LIN {X 0,Y 566.188,Z 287.454,A -85,B 0,C 180,E1 -2641.075,E2 -2641.075} C_VEL
LIN {X 0,Y 566.21,Z 287.455,A -85,B 0,C 180,E1 -2643.733,E2 -2643.733} C_VEL
LIN {X 0,Y 566.179,Z 287.455,A -85,B 0,C 180,E1 -2646.57,E2 -2646.57} C_VEL
LIN {X 0,Y 566.211,Z 287.456,A -85,B 0,C 180,E1 -2649.685,E2 -2649.685} C_VEL
LIN {X 0,Y 566.196,Z 287.452,A -85,B 0,C 180,E1 -2652.916,E2 -2652.916} C_VEL
LIN {X 0,Y 566.193,Z 287.458,A -85,B 0,C 180,E1 -2656.048,E2 -2656.048} C_VEL
LIN {X 0,Y 566.204,Z 287.45,A -85,B 0,C 180,E1 -2658.863,E2 -2658.863} C_VEL
LIN {X 0,Y 566.181,Z 287.46,A -85,B 0,C 180,E1 -2661.636,E2 -2661.636} C_VEL
LIN {X 0,Y 566.158,Z 287.457,A -85,B 0,C 180,E1 -2664.307,E2 -2664.307} C_VEL
LIN {X 0,Y 566.198,Z 287.45,A -85,B 0,C 180,E1 -2666.896,E2 -2666.896} C_VEL
LIN {X 0,Y 566.174,Z 287.46,A -85,B 0,C 180,E1 -2669.406,E2 -2669.406} C_VEL
LIN {X 0,Y 566.221,Z 287.451,A -85,B 0,C 180,E1 -2671.858,E2 -2671.858} C_VEL
LIN {X 0,Y 566.204,Z 287.45,A -85,B 0,C 180,E1 -2674.25,E2 -2674.25} C_VEL
LIN {X 0,Y 566.164,Z 287.456,A -85,B 0,C 180,E1 -2676.717,E2 -2676.717} C_VEL
LIN {X 0,Y 566.211,Z 287.454,A -85,B 0,C 180,E1 -2679.662,E2 -2679.662} C_VEL
LIN {X 0,Y 566.191,Z 287.449,A -85,B 0,C 180,E1 -2682.668,E2 -2682.668} C_VEL
LIN {X 0,Y 566.224,Z 287.454,A -85,B 0,C 180,E1 -2685.626,E2 -2685.626} C_VEL
LIN {X 0,Y 566.266,Z 287.442,A -85,B 0,C 180,E1 -2688.654,E2 -2688.654} C_VEL
LIN {X 0,Y 566.238,Z 287.452,A -85,B 0,C 180,E1 -2691.434,E2 -2691.434} C_VEL
LIN {X 0,Y 566.25,Z 287.444,A -85,B 0,C 180,E1 -2694.301,E2 -2694.301} C_VEL
LIN {X 0,Y 566.265,Z 287.443,A -85,B 0,C 180,E1 -2697.866,E2 -2697.866} C_VEL
LIN {X 0,Y 566.299,Z 287.436,A -85,B 0,C 180,E1 -2700.711,E2 -2700.711} C_VEL
LIN {X 0,Y 566.27,Z 287.445,A -85,B 0,C 180,E1 -2702.845,E2 -2702.845} C_VEL
LIN {X 0,Y 566.249,Z 287.447,A -85,B 0,C 180,E1 -2705.698,E2 -2705.698} C_VEL
LIN {X 0,Y 566.224,Z 287.448,A -85,B 0,C 180,E1 -2708.565,E2 -2708.565} C_VEL
LIN {X 0,Y 566.24,Z 287.448,A -85,B 0,C 180,E1 -2711.454,E2 -2711.454} C_VEL
LIN {X 0,Y 566.223,Z 287.451,A -85,B 0,C 180,E1 -2714.507,E2 -2714.507} C_VEL
LIN {X 0,Y 566.189,Z 287.454,A -85,B 0,C 180,E1 -2717.331,E2 -2717.331} C_VEL
LIN {X 0,Y 566.209,Z 287.448,A -85,B 0,C 180,E1 -2720.337,E2 -2720.337} C_VEL
LIN {X 0,Y 566.179,Z 287.456,A -85,B 0,C 180,E1 -2723.404,E2 -2723.404} C_VEL
LIN {X 0,Y 566.204,Z 287.449,A -85,B 0,C 180,E1 -2725.749,E2 -2725.749} C_VEL
LIN {X 0,Y 566.201,Z 287.449,A -85,B 0,C 180,E1 -2727.497,E2 -2727.497} C_VEL
LIN {X 0,Y 565.527,Z 287.533,A -85,B 0,C 180,E1 -2728.091,E2 -2728.091} C_VEL
LIN {X 0,Y 562.664,Z 287.897,A -85,B 0,C 180,E1 -2729.054,E2 -2729.054} C_VEL
LIN {X 0,Y 560.253,Z 288.195,A -85,B 0,C 180,E1 -2729.83,E2 -2729.83} C_VEL
LIN {X 0,Y 559.224,Z 288.324,A -85,B 0,C 180,E1 -2730.429,E2 -2730.429} C_VEL
LIN {X 0,Y 559.143,Z 288.332,A -85,B 0,C 180,E1 -2730.631,E2 -2730.631} C_VEL
LIN {X 0,Y 559.168,Z 288.325,A -85,B 0,C 180,E1 -2733.574,E2 -2733.574} C_VEL
LIN {X 0,Y 559.16,Z 288.332,A -85,B 0,C 180,E1 -2736.449,E2 -2736.449} C_VEL
LIN {X 0,Y 559.169,Z 288.332,A -85,B 0,C 180,E1 -2738.934,E2 -2738.934} C_VEL
LIN {X 0,Y 559.183,Z 288.324,A -85,B 0,C 180,E1 -2741.768,E2 -2741.768} C_VEL
LIN {X 0,Y 559.131,Z 288.338,A -85,B 0,C 180,E1 -2744.739,E2 -2744.739} C_VEL
LIN {X 0,Y 559.156,Z 288.322,A -85,B 0,C 180,E1 -2747.257,E2 -2747.257} C_VEL
LIN {X 0,Y 559.178,Z 288.326,A -85,B 0,C 180,E1 -2750.135,E2 -2750.135} C_VEL
LIN {X 0,Y 559.139,Z 288.334,A -85,B 0,C 180,E1 -2752.893,E2 -2752.893} C_VEL
LIN {X 0,Y 559.153,Z 288.324,A -85,B 0,C 180,E1 -2755.557,E2 -2755.557} C_VEL
LIN {X 0,Y 559.166,Z 288.333,A -85,B 0,C 180,E1 -2758.138,E2 -2758.138} C_VEL
LIN {X 0,Y 559.138,Z 288.335,A -85,B 0,C 180,E1 -2760.647,E2 -2760.647} C_VEL
LIN {X 0,Y 559.177,Z 288.327,A -85,B 0,C 180,E1 -2763.17,E2 -2763.17} C_VEL
LIN {X 0,Y 559.152,Z 288.33,A -85,B 0,C 180,E1 -2765.495,E2 -2765.495} C_VEL
LIN {X 0,Y 559.167,Z 288.333,A -85,B 0,C 180,E1 -2768.624,E2 -2768.624} C_VEL
LIN {X 0,Y 559.167,Z 288.329,A -85,B 0,C 180,E1 -2770.927,E2 -2770.927} C_VEL
LIN {X 0,Y 559.164,Z 288.334,A -85,B 0,C 180,E1 -2773.948,E2 -2773.948} C_VEL
LIN {X 0,Y 559.169,Z 288.337,A -85,B 0,C 180,E1 -2776.184,E2 -2776.184} C_VEL
LIN {X 0,Y 559.193,Z 288.325,A -85,B 0,C 180,E1 -2779.134,E2 -2779.134} C_VEL
LIN {X 0,Y 559.201,Z 288.333,A -85,B 0,C 180,E1 -2782.054,E2 -2782.054} C_VEL
LIN {X 0,Y 559.251,Z 288.318,A -85,B 0,C 180,E1 -2784.953,E2 -2784.953} C_VEL
LIN {X 0,Y 559.254,Z 288.325,A -85,B 0,C 180,E1 -2787.839,E2 -2787.839} C_VEL
LIN {X 0,Y 559.27,Z 288.317,A -85,B 0,C 180,E1 -2790.72,E2 -2790.72} C_VEL
LIN {X 0,Y 559.235,Z 288.32,A -85,B 0,C 180,E1 -2792.881,E2 -2792.881} C_VEL
LIN {X 0,Y 559.229,Z 288.328,A -85,B 0,C 180,E1 -2795.77,E2 -2795.77} C_VEL
LIN {X 0,Y 559.184,Z 288.327,A -85,B 0,C 180,E1 -2798.674,E2 -2798.674} C_VEL
LIN {X 0,Y 559.202,Z 288.33,A -85,B 0,C 180,E1 -2801.6,E2 -2801.6} C_VEL
LIN {X 0,Y 559.196,Z 288.325,A -85,B 0,C 180,E1 -2804.595,E2 -2804.595} C_VEL
LIN {X 0,Y 559.159,Z 288.336,A -85,B 0,C 180,E1 -2807.556,E2 -2807.556} C_VEL
LIN {X 0,Y 559.168,Z 288.336,A -85,B 0,C 180,E1 -2809.837,E2 -2809.837} C_VEL
LIN {X 0,Y 559.137,Z 288.335,A -85,B 0,C 180,E1 -2812.152,E2 -2812.152} C_VEL
LIN {X 0,Y 559.175,Z 288.33,A -85,B 0,C 180,E1 -2815.187,E2 -2815.187} C_VEL
LIN {X 0,Y 559.189,Z 288.332,A -85,B 0,C 180,E1 -2817.711,E2 -2817.711} C_VEL
LIN {X 0,Y 559.157,Z 288.33,A -85,B 0,C 180,E1 -2821.018,E2 -2821.018} C_VEL
LIN {X 0,Y 559.171,Z 288.325,A -85,B 0,C 180,E1 -2823.951,E2 -2823.951} C_VEL
LIN {X 0,Y 559.162,Z 288.327,A -85,B 0,C 180,E1 -2826.448,E2 -2826.448} C_VEL
LIN {X 0,Y 559.17,Z 288.329,A -85,B 0,C 180,E1 -2828.933,E2 -2828.933} C_VEL
LIN {X 0,Y 559.184,Z 288.322,A -85,B 0,C 180,E1 -2831.767,E2 -2831.767} C_VEL
LIN {X 0,Y 559.131,Z 288.331,A -85,B 0,C 180,E1 -2834.739,E2 -2834.739} C_VEL
LIN {X 0,Y 559.168,Z 288.328,A -85,B 0,C 180,E1 -2837.862,E2 -2837.862} C_VEL
LIN {X 0,Y 559.177,Z 288.325,A -85,B 0,C 180,E1 -2840.135,E2 -2840.135} C_VEL
LIN {X 0,Y 559.138,Z 288.335,A -85,B 0,C 180,E1 -2842.892,E2 -2842.892} C_VEL
LIN {X 0,Y 559.153,Z 288.332,A -85,B 0,C 180,E1 -2845.556,E2 -2845.556} C_VEL
LIN {X 0,Y 559.161,Z 288.328,A -85,B 0,C 180,E1 -2848.138,E2 -2848.138} C_VEL
LIN {X 0,Y 559.148,Z 288.331,A -85,B 0,C 180,E1 -2850.647,E2 -2850.647} C_VEL
LIN {X 0,Y 559.161,Z 288.334,A -85,B 0,C 180,E1 -2853.172,E2 -2853.172} C_VEL
LIN {X 0,Y 559.147,Z 288.334,A -85,B 0,C 180,E1 -2855.495,E2 -2855.495} C_VEL
LIN {X 0,Y 559.166,Z 288.33,A -85,B 0,C 180,E1 -2858.624,E2 -2858.624} C_VEL
LIN {X 0,Y 559.161,Z 288.332,A -85,B 0,C 180,E1 -2860.926,E2 -2860.926} C_VEL
LIN {X 0,Y 559.161,Z 288.328,A -85,B 0,C 180,E1 -2863.948,E2 -2863.948} C_VEL
LIN {X 0,Y 559.164,Z 288.328,A -85,B 0,C 180,E1 -2866.184,E2 -2866.184} C_VEL
LIN {X 0,Y 559.2,Z 288.323,A -85,B 0,C 180,E1 -2869.134,E2 -2869.134} C_VEL
LIN {X 0,Y 559.196,Z 288.321,A -85,B 0,C 180,E1 -2872.054,E2 -2872.054} C_VEL
LIN {X 0,Y 559.249,Z 288.325,A -85,B 0,C 180,E1 -2874.954,E2 -2874.954} C_VEL
LIN {X 0,Y 559.238,Z 288.316,A -85,B 0,C 180,E1 -2877.84,E2 -2877.84} C_VEL
LIN {X 0,Y 559.269,Z 288.317,A -85,B 0,C 180,E1 -2880.72,E2 -2880.72} C_VEL
LIN {X 0,Y 559.234,Z 288.326,A -85,B 0,C 180,E1 -2882.882,E2 -2882.882} C_VEL
LIN {X 0,Y 559.219,Z 288.32,A -85,B 0,C 180,E1 -2885.771,E2 -2885.771} C_VEL
LIN {X 0,Y 559.193,Z 288.327,A -85,B 0,C 180,E1 -2888.675,E2 -2888.675} C_VEL
LIN {X 0,Y 559.2,Z 288.321,A -85,B 0,C 180,E1 -2891.601,E2 -2891.601} C_VEL
LIN {X 0,Y 559.19,Z 288.333,A -85,B 0,C 180,E1 -2894.596,E2 -2894.596} C_VEL
LIN {X 0,Y 559.151,Z 288.325,A -85,B 0,C 180,E1 -2897.558,E2 -2897.558} C_VEL
LIN {X 0,Y 559.166,Z 288.324,A -85,B 0,C 180,E1 -2899.838,E2 -2899.838} C_VEL
LIN {X 0,Y 559.133,Z 288.335,A -85,B 0,C 180,E1 -2902.154,E2 -2902.154} C_VEL
LIN {X 0,Y 559.167,Z 288.325,A -85,B 0,C 180,E1 -2905.299,E2 -2905.299} C_VEL
LIN {X 0,Y 559.185,Z 288.322,A -85,B 0,C 180,E1 -2907.712,E2 -2907.712} C_VEL
LIN {X 0,Y 559.146,Z 288.336,A -85,B 0,C 180,E1 -2910.184,E2 -2910.184} C_VEL
LIN {X 0,Y 559.146,Z 288.331,A -85,B 0,C 180,E1 -2912.716,E2 -2912.716} C_VEL
LIN {X 0,Y 559.123,Z 288.331,A -85,B 0,C 180,E1 -2915.325,E2 -2915.325} C_VEL
LIN {X 0,Y 559.127,Z 288.338,A -85,B 0,C 180,E1 -2918.018,E2 -2918.018} C_VEL
LIN {X 0,Y 559.152,Z 288.33,A -85,B 0,C 180,E1 -2920.813,E2 -2920.813} C_VEL
LIN {X 0,Y 559.142,Z 288.33,A -85,B 0,C 180,E1 -2923.197,E2 -2923.197} C_VEL
LIN {X 0,Y 559.136,Z 288.339,A -85,B 0,C 180,E1 -2926.267,E2 -2926.267} C_VEL
LIN {X 0,Y 559.152,Z 288.325,A -85,B 0,C 180,E1 -2929.188,E2 -2929.188} C_VEL
LIN {X 0,Y 559.127,Z 288.341,A -85,B 0,C 180,E1 -2931.983,E2 -2931.983} C_VEL
LIN {X 0,Y 559.127,Z 288.333,A -85,B 0,C 180,E1 -2934.788,E2 -2934.788} C_VEL
LIN {X 0,Y 559.154,Z 288.33,A -85,B 0,C 180,E1 -2937.365,E2 -2937.365} C_VEL
LIN {X 0,Y 559.146,Z 288.338,A -85,B 0,C 180,E1 -2940.144,E2 -2940.144} C_VEL
LIN {X 0,Y 559.163,Z 288.332,A -85,B 0,C 180,E1 -2943.175,E2 -2943.175} C_VEL
LIN {X 0,Y 559.212,Z 288.44,A -85,B 0,C 180,E1 -2944.807,E2 -2944.807} C_VEL
LIN {X 0,Y 559.948,Z 294.047,A -85,B 0,C 180,E1 -2945.927,E2 -2945.927} C_VEL
LIN {X 0,Y 559.68,Z 309.675,A -85,B 0,C 180,E1 -2948.838,E2 -2948.838} C_VEL
LIN {X 0,Y 559.517,Z 326.41,A -85,B 0,C 180,E1 -2951.888,E2 -2951.888} C_VEL
LIN {X 0,Y 559.299,Z 343.133,A -85,B 0,C 180,E1 -2954.905,E2 -2954.905} C_VEL
LIN {X 0,Y 559.262,Z 348.266,A -85,B 0,C 180,E1 -2955.792,E2 -2955.792} C_VEL
LIN {X 0,Y 559.602,Z 350.542,A -85,B 0,C 180,E1 -2955.868,E2 -2955.868} C_VEL
LIN {X 0,Y 560.311,Z 356.112,A -85,B 0,C 180,E1 -2955.959,E2 -2955.959} C_VEL
LIN {X 0,Y 560.037,Z 454.578,A -85,B 0,C 180,E1 -2957.245,E2 -2957.245} C_VEL
LIN {X 0,Y 559.976,Z 465.719,A -85,B 0,C 180,E1 -2957.497,E2 -2957.497} C_VEL
LIN {X 0,Y 559.814,Z 478.172,A -85,B 0,C 180,E1 -2957.908,E2 -2957.908} C_VEL
LIN {X 0,Y 559.678,Z 490.904,A -85,B 0,C 180,E1 -2958.503,E2 -2958.503} C_VEL
LIN {X 0,Y 559.509,Z 501.475,A -85,B 0,C 180,E1 -2959.14,E2 -2959.14} C_VEL
LIN {X 0,Y 559.379,Z 510.174,A -85,B 0,C 180,E1 -2959.778,E2 -2959.778} C_VEL
LIN {X 0,Y 559.274,Z 517.542,A -85,B 0,C 180,E1 -2960.416,E2 -2960.416} C_VEL
LIN {X 0,Y 559.137,Z 524.73,A -85,B 0,C 180,E1 -2961.143,E2 -2961.143} C_VEL
LIN {X 0,Y 559.052,Z 532.276,A -85,B 0,C 180,E1 -2962.052,E2 -2962.052} C_VEL
LIN {X 0,Y 558.934,Z 538.681,A -85,B 0,C 180,E1 -2962.976,E2 -2962.976} C_VEL
LIN {X 0,Y 558.909,Z 543.8,A -85,B 0,C 180,E1 -2963.864,E2 -2963.864} C_VEL
LIN {X 0,Y 558.798,Z 548.897,A -85,B 0,C 180,E1 -2964.949,E2 -2964.949} C_VEL
LIN {X 0,Y 558.843,Z 552.853,A -85,B 0,C 180,E1 -2966.034,E2 -2966.034} C_VEL
LIN {X 0,Y 558.799,Z 555.774,A -85,B 0,C 180,E1 -2967.116,E2 -2967.116} C_VEL
LIN {X 0,Y 558.746,Z 558.196,A -85,B 0,C 180,E1 -2968.559,E2 -2968.559} C_VEL
LIN {X 0,Y 558.741,Z 558.78,A -85,B 0,C 180,E1 -2969.279,E2 -2969.279} C_VEL
LIN {X 0,Y 558.741,Z 558.78,A -85,B 0,C 180,E1 -2970.721,E2 -2970.721} C_VEL
LIN {X 0,Y 558.746,Z 558.196,A -85,B 0,C 180,E1 -2971.441,E2 -2971.441} C_VEL
LIN {X 0,Y 558.799,Z 555.774,A -85,B 0,C 180,E1 -2972.884,E2 -2972.884} C_VEL
LIN {X 0,Y 558.843,Z 552.853,A -85,B 0,C 180,E1 -2973.966,E2 -2973.966} C_VEL
LIN {X 0,Y 558.798,Z 548.897,A -85,B 0,C 180,E1 -2975.051,E2 -2975.051} C_VEL
LIN {X 0,Y 558.91,Z 543.8,A -85,B 0,C 180,E1 -2976.136,E2 -2976.136} C_VEL
LIN {X 0,Y 558.974,Z 537.416,A -85,B 0,C 180,E1 -2977.223,E2 -2977.223} C_VEL
LIN {X 0,Y 559.093,Z 529.505,A -85,B 0,C 180,E1 -2978.312,E2 -2978.312} C_VEL
LIN {X 0,Y 559.209,Z 521.359,A -85,B 0,C 180,E1 -2979.221,E2 -2979.221} C_VEL
LIN {X 0,Y 559.33,Z 511.306,A -85,B 0,C 180,E1 -2980.131,E2 -2980.131} C_VEL
LIN {X 0,Y 559.499,Z 502.823,A -85,B 0,C 180,E1 -2980.769,E2 -2980.769} C_VEL
LIN {X 0,Y 559.631,Z 493.792,A -85,B 0,C 180,E1 -2981.335,E2 -2981.335} C_VEL
LIN {X 0,Y 559.768,Z 483.593,A -85,B 0,C 180,E1 -2981.854,E2 -2981.854} C_VEL
LIN {X 0,Y 559.863,Z 474.329,A -85,B 0,C 180,E1 -2982.229,E2 -2982.229} C_VEL
LIN {X 0,Y 559.966,Z 463.971,A -85,B 0,C 180,E1 -2982.549,E2 -2982.549} C_VEL
LIN {X 0,Y 560.068,Z 453.247,A -85,B 0,C 180,E1 -2982.777,E2 -2982.777} C_VEL
LIN {X 0,Y 560.236,Z 354.323,A -85,B 0,C 180,E1 -2984.066,E2 -2984.066} C_VEL
LIN {X 0,Y 559.275,Z 348.595,A -85,B 0,C 180,E1 -2984.184,E2 -2984.184} C_VEL
LIN {X 0,Y 559.225,Z 347.169,A -85,B 0,C 180,E1 -2984.371,E2 -2984.371} C_VEL
LIN {X 0,Y 559.444,Z 330.904,A -85,B 0,C 180,E1 -2987.302,E2 -2987.302} C_VEL
LIN {X 0,Y 559.662,Z 313.862,A -85,B 0,C 180,E1 -2990.393,E2 -2990.393} C_VEL
LIN {X 0,Y 559.864,Z 298.427,A -85,B 0,C 180,E1 -2993.255,E2 -2993.255} C_VEL
LIN {X 0,Y 559.822,Z 291.989,A -85,B 0,C 180,E1 -2994.473,E2 -2994.473} C_VEL
LIN {X 0,Y 559.189,Z 288.353,A -85,B 0,C 180,E1 -2995.251,E2 -2995.251} C_VEL
LIN {X 0,Y 559.138,Z 288.339,A -85,B 0,C 180,E1 -2997.714,E2 -2997.714} C_VEL
LIN {X 0,Y 559.151,Z 288.338,A -85,B 0,C 180,E1 -3000.182,E2 -3000.182} C_VEL
LIN {X 0,Y 559.155,Z 288.329,A -85,B 0,C 180,E1 -3002.714,E2 -3002.714} C_VEL
LIN {X 0,Y 559.121,Z 288.334,A -85,B 0,C 180,E1 -3005.324,E2 -3005.324} C_VEL
LIN {X 0,Y 559.127,Z 288.341,A -85,B 0,C 180,E1 -3008.017,E2 -3008.017} C_VEL
LIN {X 0,Y 559.152,Z 288.325,A -85,B 0,C 180,E1 -3010.812,E2 -3010.812} C_VEL
LIN {X 0,Y 559.136,Z 288.339,A -85,B 0,C 180,E1 -3013.733,E2 -3013.733} C_VEL
LIN {X 0,Y 559.142,Z 288.33,A -85,B 0,C 180,E1 -3016.803,E2 -3016.803} C_VEL
LIN {X 0,Y 559.171,Z 288.328,A -85,B 0,C 180,E1 -3019.188,E2 -3019.188} C_VEL
LIN {X 0,Y 559.127,Z 288.338,A -85,B 0,C 180,E1 -3021.982,E2 -3021.982} C_VEL
LIN {X 0,Y 559.127,Z 288.331,A -85,B 0,C 180,E1 -3024.786,E2 -3024.786} C_VEL
LIN {X 0,Y 559.148,Z 288.332,A -85,B 0,C 180,E1 -3027.364,E2 -3027.364} C_VEL
LIN {X 0,Y 559.141,Z 288.333,A -85,B 0,C 180,E1 -3030.142,E2 -3030.142} C_VEL
LIN {X 0,Y 559.163,Z 288.327,A -85,B 0,C 180,E1 -3033.097,E2 -3033.097} C_VEL
LIN {X 0,Y 559.148,Z 288.336,A -85,B 0,C 180,E1 -3035.494,E2 -3035.494} C_VEL
LIN {X 0,Y 559.169,Z 288.326,A -85,B 0,C 180,E1 -3038.623,E2 -3038.623} C_VEL
LIN {X 0,Y 559.161,Z 288.326,A -85,B 0,C 180,E1 -3040.926,E2 -3040.926} C_VEL
LIN {X 0,Y 559.161,Z 288.33,A -85,B 0,C 180,E1 -3043.947,E2 -3043.947} C_VEL
LIN {X 0,Y 559.165,Z 288.327,A -85,B 0,C 180,E1 -3046.184,E2 -3046.184} C_VEL
LIN {X 0,Y 559.2,Z 288.327,A -85,B 0,C 180,E1 -3049.133,E2 -3049.133} C_VEL
LIN {X 0,Y 559.2,Z 288.321,A -85,B 0,C 180,E1 -3052.053,E2 -3052.053} C_VEL
LIN {X 0,Y 559.249,Z 288.321,A -85,B 0,C 180,E1 -3054.953,E2 -3054.953} C_VEL
LIN {X 0,Y 559.237,Z 288.318,A -85,B 0,C 180,E1 -3057.839,E2 -3057.839} C_VEL
LIN {X 0,Y 559.268,Z 288.311,A -85,B 0,C 180,E1 -3060.72,E2 -3060.72} C_VEL
LIN {X 0,Y 559.236,Z 288.321,A -85,B 0,C 180,E1 -3062.881,E2 -3062.881} C_VEL
LIN {X 0,Y 559.218,Z 288.322,A -85,B 0,C 180,E1 -3065.77,E2 -3065.77} C_VEL
LIN {X 0,Y 559.182,Z 288.326,A -85,B 0,C 180,E1 -3068.674,E2 -3068.674} C_VEL
LIN {X 0,Y 559.198,Z 288.324,A -85,B 0,C 180,E1 -3071.6,E2 -3071.6} C_VEL
LIN {X 0,Y 559.188,Z 288.328,A -85,B 0,C 180,E1 -3074.595,E2 -3074.595} C_VEL
LIN {X 0,Y 559.149,Z 288.328,A -85,B 0,C 180,E1 -3077.557,E2 -3077.557} C_VEL
LIN {X 0,Y 559.164,Z 288.324,A -85,B 0,C 180,E1 -3079.837,E2 -3079.837} C_VEL
LIN {X 0,Y 559.132,Z 288.331,A -85,B 0,C 180,E1 -3082.153,E2 -3082.153} C_VEL
LIN {X 0,Y 559.168,Z 288.33,A -85,B 0,C 180,E1 -3085.187,E2 -3085.187} C_VEL
LIN {X 0,Y 559.181,Z 288.322,A -85,B 0,C 180,E1 -3087.712,E2 -3087.712} C_VEL
LIN {X 0,Y 559.143,Z 288.332,A -85,B 0,C 180,E1 -3090.631,E2 -3090.631} C_VEL
LIN {X 0,Y 558.481,Z 288.418,A -85,B 0,C 180,E1 -3091.233,E2 -3091.233} C_VEL
LIN {X 0,Y 555.617,Z 288.773,A -85,B 0,C 180,E1 -3092.209,E2 -3092.209} C_VEL
LIN {X 0,Y 553.206,Z 289.074,A -85,B 0,C 180,E1 -3092.995,E2 -3092.995} C_VEL
LIN {X 0,Y 552.187,Z 289.195,A -85,B 0,C 180,E1 -3093.601,E2 -3093.601} C_VEL
LIN {X 0,Y 552.114,Z 289.203,A -85,B 0,C 180,E1 -3093.807,E2 -3093.807} C_VEL
LIN {X 0,Y 552.102,Z 289.217,A -85,B 0,C 180,E1 -3096.747,E2 -3096.747} C_VEL
LIN {X 0,Y 552.126,Z 289.203,A -85,B 0,C 180,E1 -3099.527,E2 -3099.527} C_VEL
LIN {X 0,Y 552.122,Z 289.21,A -85,B 0,C 180,E1 -3102.426,E2 -3102.426} C_VEL
LIN {X 0,Y 552.091,Z 289.207,A -85,B 0,C 180,E1 -3105.563,E2 -3105.563} C_VEL
LIN {X 0,Y 552.132,Z 289.205,A -85,B 0,C 180,E1 -3108.676,E2 -3108.676} C_VEL
LIN {X 0,Y 552.112,Z 289.207,A -85,B 0,C 180,E1 -3111.412,E2 -3111.412} C_VEL
LIN {X 0,Y 552.106,Z 289.211,A -85,B 0,C 180,E1 -3114.159,E2 -3114.159} C_VEL
LIN {X 0,Y 552.123,Z 289.209,A -85,B 0,C 180,E1 -3116.816,E2 -3116.816} C_VEL
LIN {X 0,Y 552.102,Z 289.207,A -85,B 0,C 180,E1 -3119.391,E2 -3119.391} C_VEL
LIN {X 0,Y 552.121,Z 289.206,A -85,B 0,C 180,E1 -3121.903,E2 -3121.903} C_VEL
LIN {X 0,Y 552.152,Z 289.207,A -85,B 0,C 180,E1 -3124.649,E2 -3124.649} C_VEL
LIN {X 0,Y 552.091,Z 289.21,A -85,B 0,C 180,E1 -3127.55,E2 -3127.55} C_VEL
LIN {X 0,Y 552.153,Z 289.206,A -85,B 0,C 180,E1 -3130.675,E2 -3130.675} C_VEL
LIN {X 0,Y 552.114,Z 289.21,A -85,B 0,C 180,E1 -3133.738,E2 -3133.738} C_VEL
LIN {X 0,Y 552.132,Z 289.212,A -85,B 0,C 180,E1 -3136.005,E2 -3136.005} C_VEL
LIN {X 0,Y 552.16,Z 289.202,A -85,B 0,C 180,E1 -3138.994,E2 -3138.994} C_VEL
LIN {X 0,Y 552.155,Z 289.21,A -85,B 0,C 180,E1 -3141.952,E2 -3141.952} C_VEL
LIN {X 0,Y 552.226,Z 289.194,A -85,B 0,C 180,E1 -3144.889,E2 -3144.889} C_VEL
LIN {X 0,Y 552.224,Z 289.2,A -85,B 0,C 180,E1 -3147.812,E2 -3147.812} C_VEL
LIN {X 0,Y 552.24,Z 289.193,A -85,B 0,C 180,E1 -3150.729,E2 -3150.729} C_VEL
LIN {X 0,Y 552.202,Z 289.197,A -85,B 0,C 180,E1 -3152.918,E2 -3152.918} C_VEL
LIN {X 0,Y 552.199,Z 289.205,A -85,B 0,C 180,E1 -3155.844,E2 -3155.844} C_VEL
LIN {X 0,Y 552.156,Z 289.202,A -85,B 0,C 180,E1 -3158.786,E2 -3158.786} C_VEL
LIN {X 0,Y 552.159,Z 289.209,A -85,B 0,C 180,E1 -3161.75,E2 -3161.75} C_VEL
LIN {X 0,Y 552.133,Z 289.205,A -85,B 0,C 180,E1 -3164.748,E2 -3164.748} C_VEL
LIN {X 0,Y 552.111,Z 289.216,A -85,B 0,C 180,E1 -3167.788,E2 -3167.788} C_VEL
LIN {X 0,Y 552.127,Z 289.209,A -85,B 0,C 180,E1 -3170.101,E2 -3170.101} C_VEL
LIN {X 0,Y 552.091,Z 289.21,A -85,B 0,C 180,E1 -3172.45,E2 -3172.45} C_VEL
LIN {X 0,Y 552.152,Z 289.207,A -85,B 0,C 180,E1 -3175.351,E2 -3175.351} C_VEL
LIN {X 0,Y 552.121,Z 289.206,A -85,B 0,C 180,E1 -3178.097,E2 -3178.097} C_VEL
LIN {X 0,Y 552.102,Z 289.207,A -85,B 0,C 180,E1 -3180.609,E2 -3180.609} C_VEL
LIN {X 0,Y 552.123,Z 289.209,A -85,B 0,C 180,E1 -3183.184,E2 -3183.184} C_VEL
LIN {X 0,Y 552.106,Z 289.211,A -85,B 0,C 180,E1 -3185.841,E2 -3185.841} C_VEL
LIN {X 0,Y 552.118,Z 289.209,A -85,B 0,C 180,E1 -3189.062,E2 -3189.062} C_VEL
LIN {X 0,Y 552.132,Z 289.203,A -85,B 0,C 180,E1 -3191.444,E2 -3191.444} C_VEL
LIN {X 0,Y 552.088,Z 289.207,A -85,B 0,C 180,E1 -3194.532,E2 -3194.532} C_VEL
LIN {X 0,Y 552.122,Z 289.21,A -85,B 0,C 180,E1 -3197.584,E2 -3197.584} C_VEL
LIN {X 0,Y 552.126,Z 289.203,A -85,B 0,C 180,E1 -3200.473,E2 -3200.473} C_VEL
LIN {X 0,Y 552.105,Z 289.215,A -85,B 0,C 180,E1 -3203.315,E2 -3203.315} C_VEL
LIN {X 0,Y 552.131,Z 289.202,A -85,B 0,C 180,E1 -3205.94,E2 -3205.94} C_VEL
LIN {X 0,Y 552.108,Z 289.208,A -85,B 0,C 180,E1 -3208.54,E2 -3208.54} C_VEL
LIN {X 0,Y 552.117,Z 289.207,A -85,B 0,C 180,E1 -3211.437,E2 -3211.437} C_VEL
LIN {X 0,Y 552.119,Z 289.204,A -85,B 0,C 180,E1 -3214.356,E2 -3214.356} C_VEL
LIN {X 0,Y 552.1,Z 289.212,A -85,B 0,C 180,E1 -3216.758,E2 -3216.758} C_VEL
LIN {X 0,Y 552.117,Z 289.21,A -85,B 0,C 180,E1 -3219.12,E2 -3219.12} C_VEL
LIN {X 0,Y 552.121,Z 289.205,A -85,B 0,C 180,E1 -3221.445,E2 -3221.445} C_VEL
LIN {X 0,Y 552.111,Z 289.206,A -85,B 0,C 180,E1 -3223.738,E2 -3223.738} C_VEL
LIN {X 0,Y 552.126,Z 289.204,A -85,B 0,C 180,E1 -3226.005,E2 -3226.005} C_VEL
LIN {X 0,Y 552.168,Z 289.201,A -85,B 0,C 180,E1 -3228.994,E2 -3228.994} C_VEL
LIN {X 0,Y 552.15,Z 289.199,A -85,B 0,C 180,E1 -3231.952,E2 -3231.952} C_VEL
LIN {X 0,Y 552.223,Z 289.201,A -85,B 0,C 180,E1 -3234.889,E2 -3234.889} C_VEL
LIN {X 0,Y 552.211,Z 289.191,A -85,B 0,C 180,E1 -3237.812,E2 -3237.812} C_VEL
LIN {X 0,Y 552.239,Z 289.192,A -85,B 0,C 180,E1 -3240.73,E2 -3240.73} C_VEL
LIN {X 0,Y 552.2,Z 289.202,A -85,B 0,C 180,E1 -3242.919,E2 -3242.919} C_VEL
LIN {X 0,Y 552.189,Z 289.196,A -85,B 0,C 180,E1 -3245.844,E2 -3245.844} C_VEL
LIN {X 0,Y 552.161,Z 289.2,A -85,B 0,C 180,E1 -3248.786,E2 -3248.786} C_VEL
LIN {X 0,Y 552.155,Z 289.198,A -85,B 0,C 180,E1 -3251.751,E2 -3251.751} C_VEL
LIN {X 0,Y 552.127,Z 289.21,A -85,B 0,C 180,E1 -3254.749,E2 -3254.749} C_VEL
LIN {X 0,Y 552.102,Z 289.204,A -85,B 0,C 180,E1 -3257.789,E2 -3257.789} C_VEL
LIN {X 0,Y 552.126,Z 289.204,A -85,B 0,C 180,E1 -3260.102,E2 -3260.102} C_VEL
LIN {X 0,Y 552.084,Z 289.218,A -85,B 0,C 180,E1 -3262.452,E2 -3262.452} C_VEL
LIN {X 0,Y 552.147,Z 289.199,A -85,B 0,C 180,E1 -3265.351,E2 -3265.351} C_VEL
LIN {X 0,Y 552.119,Z 289.206,A -85,B 0,C 180,E1 -3268.098,E2 -3268.098} C_VEL
LIN {X 0,Y 552.095,Z 289.214,A -85,B 0,C 180,E1 -3270.61,E2 -3270.61} C_VEL
LIN {X 0,Y 552.1,Z 289.205,A -85,B 0,C 180,E1 -3273.187,E2 -3273.187} C_VEL
LIN {X 0,Y 552.08,Z 289.212,A -85,B 0,C 180,E1 -3275.844,E2 -3275.844} C_VEL
LIN {X 0,Y 552.112,Z 289.209,A -85,B 0,C 180,E1 -3278.59,E2 -3278.59} C_VEL
LIN {X 0,Y 552.125,Z 289.205,A -85,B 0,C 180,E1 -3281.446,E2 -3281.446} C_VEL
LIN {X 0,Y 552.089,Z 289.213,A -85,B 0,C 180,E1 -3284.532,E2 -3284.532} C_VEL
LIN {X 0,Y 552.126,Z 289.207,A -85,B 0,C 180,E1 -3287.586,E2 -3287.586} C_VEL
LIN {X 0,Y 552.126,Z 289.208,A -85,B 0,C 180,E1 -3290.474,E2 -3290.474} C_VEL
LIN {X 0,Y 552.096,Z 289.209,A -85,B 0,C 180,E1 -3293.319,E2 -3293.319} C_VEL
LIN {X 0,Y 552.124,Z 289.213,A -85,B 0,C 180,E1 -3295.94,E2 -3295.94} C_VEL
LIN {X 0,Y 552.119,Z 289.209,A -85,B 0,C 180,E1 -3298.541,E2 -3298.541} C_VEL
LIN {X 0,Y 552.104,Z 289.212,A -85,B 0,C 180,E1 -3301.443,E2 -3301.443} C_VEL
LIN {X 0,Y 552.126,Z 289.212,A -85,B 0,C 180,E1 -3304.356,E2 -3304.356} C_VEL
LIN {X 0,Y 552.163,Z 289.447,A -85,B 0,C 180,E1 -3304.686,E2 -3304.686} C_VEL
LIN {X 0,Y 553.01,Z 294.996,A -85,B 0,C 180,E1 -3305.805,E2 -3305.805} C_VEL
LIN {X 0,Y 552.706,Z 310.587,A -85,B 0,C 180,E1 -3308.753,E2 -3308.753} C_VEL
LIN {X 0,Y 552.501,Z 327.322,A -85,B 0,C 180,E1 -3311.842,E2 -3311.842} C_VEL
LIN {X 0,Y 552.283,Z 344.026,A -85,B 0,C 180,E1 -3314.879,E2 -3314.879} C_VEL
LIN {X 0,Y 552.236,Z 348.45,A -85,B 0,C 180,E1 -3315.622,E2 -3315.622} C_VEL
LIN {X 0,Y 553.424,Z 355.602,A -85,B 0,C 180,E1 -3315.773,E2 -3315.773} C_VEL
LIN {X 0,Y 553.139,Z 453.191,A -85,B 0,C 180,E1 -3317.06,E2 -3317.06} C_VEL
LIN {X 0,Y 553.051,Z 463.937,A -85,B 0,C 180,E1 -3317.291,E2 -3317.291} C_VEL
LIN {X 0,Y 552.925,Z 474.306,A -85,B 0,C 180,E1 -3317.615,E2 -3317.615} C_VEL
LIN {X 0,Y 552.767,Z 484.372,A -85,B 0,C 180,E1 -3318.03,E2 -3318.03} C_VEL
LIN {X 0,Y 552.636,Z 494.743,A -85,B 0,C 180,E1 -3318.575,E2 -3318.575} C_VEL
LIN {X 0,Y 552.469,Z 505.496,A -85,B 0,C 180,E1 -3319.278,E2 -3319.278} C_VEL
LIN {X 0,Y 552.272,Z 515.616,A -85,B 0,C 180,E1 -3320.108,E2 -3320.108} C_VEL
LIN {X 0,Y 552.122,Z 524.721,A -85,B 0,C 180,E1 -3321.029,E2 -3321.029} C_VEL
LIN {X 0,Y 551.984,Z 532.268,A -85,B 0,C 180,E1 -3321.949,E2 -3321.949} C_VEL
LIN {X 0,Y 551.886,Z 538.557,A -85,B 0,C 180,E1 -3322.868,E2 -3322.868} C_VEL
LIN {X 0,Y 551.836,Z 544.396,A -85,B 0,C 180,E1 -3323.902,E2 -3323.902} C_VEL
LIN {X 0,Y 551.739,Z 550.388,A -85,B 0,C 180,E1 -3325.251,E2 -3325.251} C_VEL
LIN {X 0,Y 551.75,Z 553.976,A -85,B 0,C 180,E1 -3326.349,E2 -3326.349} C_VEL
LIN {X 0,Y 551.723,Z 555.768,A -85,B 0,C 180,E1 -3327.079,E2 -3327.079} C_VEL
LIN {X 0,Y 551.645,Z 558.195,A -85,B 0,C 180,E1 -3328.54,E2 -3328.54} C_VEL
LIN {X 0,Y 551.641,Z 558.779,A -85,B 0,C 180,E1 -3329.27,E2 -3329.27} C_VEL
LIN {X 0,Y 551.641,Z 558.779,A -85,B 0,C 180,E1 -3330.73,E2 -3330.73} C_VEL
LIN {X 0,Y 551.645,Z 558.195,A -85,B 0,C 180,E1 -3331.46,E2 -3331.46} C_VEL
LIN {X 0,Y 551.723,Z 555.768,A -85,B 0,C 180,E1 -3332.921,E2 -3332.921} C_VEL
LIN {X 0,Y 551.764,Z 552.845,A -85,B 0,C 180,E1 -3334.017,E2 -3334.017} C_VEL
LIN {X 0,Y 551.723,Z 548.888,A -85,B 0,C 180,E1 -3335.116,E2 -3335.116} C_VEL
LIN {X 0,Y 551.836,Z 544.395,A -85,B 0,C 180,E1 -3336.098,E2 -3336.098} C_VEL
LIN {X 0,Y 551.886,Z 538.557,A -85,B 0,C 180,E1 -3337.132,E2 -3337.132} C_VEL
LIN {X 0,Y 551.984,Z 532.268,A -85,B 0,C 180,E1 -3338.051,E2 -3338.051} C_VEL
LIN {X 0,Y 552.122,Z 524.721,A -85,B 0,C 180,E1 -3338.971,E2 -3338.971} C_VEL
LIN {X 0,Y 552.272,Z 515.616,A -85,B 0,C 180,E1 -3339.892,E2 -3339.892} C_VEL
LIN {X 0,Y 552.489,Z 504.156,A -85,B 0,C 180,E1 -3340.814,E2 -3340.814} C_VEL
LIN {X 0,Y 552.632,Z 494.762,A -85,B 0,C 180,E1 -3341.424,E2 -3341.424} C_VEL
LIN {X 0,Y 552.794,Z 484.679,A -85,B 0,C 180,E1 -3341.955,E2 -3341.955} C_VEL
LIN {X 0,Y 552.881,Z 475.596,A -85,B 0,C 180,E1 -3342.34,E2 -3342.34} C_VEL
LIN {X 0,Y 553.054,Z 464.811,A -85,B 0,C 180,E1 -3342.685,E2 -3342.685} C_VEL
LIN {X 0,Y 553.131,Z 454.522,A -85,B 0,C 180,E1 -3342.917,E2 -3342.917} C_VEL
LIN {X 0,Y 553.343,Z 369.327,A -85,B 0,C 180,E1 -3344.049,E2 -3344.049} C_VEL
LIN {X 0,Y 553.316,Z 354.796,A -85,B 0,C 180,E1 -3344.24,E2 -3344.24} C_VEL
LIN {X 0,Y 552.236,Z 348.447,A -85,B 0,C 180,E1 -3344.378,E2 -3344.378} C_VEL
LIN {X 0,Y 552.283,Z 344.026,A -85,B 0,C 180,E1 -3345.121,E2 -3345.121} C_VEL
LIN {X 0,Y 552.501,Z 327.322,A -85,B 0,C 180,E1 -3348.158,E2 -3348.158} C_VEL
LIN {X 0,Y 552.706,Z 310.619,A -85,B 0,C 180,E1 -3351.247,E2 -3351.247} C_VEL
LIN {X 0,Y 552.99,Z 295.021,A -85,B 0,C 180,E1 -3354.196,E2 -3354.196} C_VEL
LIN {X 0,Y 552.151,Z 289.247,A -85,B 0,C 180,E1 -3355.385,E2 -3355.385} C_VEL
LIN {X 0,Y 552.088,Z 289.217,A -85,B 0,C 180,E1 -3358.099,E2 -3358.099} C_VEL
LIN {X 0,Y 552.1,Z 289.211,A -85,B 0,C 180,E1 -3360.609,E2 -3360.609} C_VEL
LIN {X 0,Y 552.114,Z 289.206,A -85,B 0,C 180,E1 -3363.185,E2 -3363.185} C_VEL
LIN {X 0,Y 552.072,Z 289.217,A -85,B 0,C 180,E1 -3365.844,E2 -3365.844} C_VEL
LIN {X 0,Y 552.113,Z 289.207,A -85,B 0,C 180,E1 -3368.588,E2 -3368.588} C_VEL
LIN {X 0,Y 552.116,Z 289.204,A -85,B 0,C 180,E1 -3371.445,E2 -3371.445} C_VEL
LIN {X 0,Y 552.088,Z 289.21,A -85,B 0,C 180,E1 -3374.531,E2 -3374.531} C_VEL
LIN {X 0,Y 552.127,Z 289.21,A -85,B 0,C 180,E1 -3377.584,E2 -3377.584} C_VEL
LIN {X 0,Y 552.125,Z 289.204,A -85,B 0,C 180,E1 -3380.472,E2 -3380.472} C_VEL
LIN {X 0,Y 552.1,Z 289.211,A -85,B 0,C 180,E1 -3383.316,E2 -3383.316} C_VEL
LIN {X 0,Y 552.098,Z 289.211,A -85,B 0,C 180,E1 -3385.937,E2 -3385.937} C_VEL
LIN {X 0,Y 552.112,Z 289.206,A -85,B 0,C 180,E1 -3388.54,E2 -3388.54} C_VEL
LIN {X 0,Y 552.119,Z 289.212,A -85,B 0,C 180,E1 -3391.437,E2 -3391.437} C_VEL
LIN {X 0,Y 552.122,Z 289.203,A -85,B 0,C 180,E1 -3394.355,E2 -3394.355} C_VEL
LIN {X 0,Y 552.09,Z 289.209,A -85,B 0,C 180,E1 -3396.757,E2 -3396.757} C_VEL
LIN {X 0,Y 552.118,Z 289.208,A -85,B 0,C 180,E1 -3399.119,E2 -3399.119} C_VEL
LIN {X 0,Y 552.119,Z 289.208,A -85,B 0,C 180,E1 -3401.444,E2 -3401.444} C_VEL
LIN {X 0,Y 552.111,Z 289.21,A -85,B 0,C 180,E1 -3403.737,E2 -3403.737} C_VEL
LIN {X 0,Y 552.128,Z 289.205,A -85,B 0,C 180,E1 -3406.004,E2 -3406.004} C_VEL
LIN {X 0,Y 552.168,Z 289.2,A -85,B 0,C 180,E1 -3408.993,E2 -3408.993} C_VEL
LIN {X 0,Y 552.154,Z 289.199,A -85,B 0,C 180,E1 -3411.951,E2 -3411.951} C_VEL
LIN {X 0,Y 552.223,Z 289.196,A -85,B 0,C 180,E1 -3414.889,E2 -3414.889} C_VEL
LIN {X 0,Y 552.21,Z 289.193,A -85,B 0,C 180,E1 -3417.811,E2 -3417.811} C_VEL
LIN {X 0,Y 552.238,Z 289.186,A -85,B 0,C 180,E1 -3420.729,E2 -3420.729} C_VEL
LIN {X 0,Y 552.202,Z 289.197,A -85,B 0,C 180,E1 -3422.918,E2 -3422.918} C_VEL
LIN {X 0,Y 552.188,Z 289.197,A -85,B 0,C 180,E1 -3425.844,E2 -3425.844} C_VEL
LIN {X 0,Y 552.153,Z 289.203,A -85,B 0,C 180,E1 -3428.785,E2 -3428.785} C_VEL
LIN {X 0,Y 552.154,Z 289.2,A -85,B 0,C 180,E1 -3431.75,E2 -3431.75} C_VEL
LIN {X 0,Y 552.126,Z 289.21,A -85,B 0,C 180,E1 -3434.748,E2 -3434.748} C_VEL
LIN {X 0,Y 552.1,Z 289.204,A -85,B 0,C 180,E1 -3437.788,E2 -3437.788} C_VEL
LIN {X 0,Y 552.123,Z 289.201,A -85,B 0,C 180,E1 -3440.101,E2 -3440.101} C_VEL
LIN {X 0,Y 552.086,Z 289.211,A -85,B 0,C 180,E1 -3442.451,E2 -3442.451} C_VEL
LIN {X 0,Y 552.144,Z 289.203,A -85,B 0,C 180,E1 -3445.351,E2 -3445.351} C_VEL
LIN {X 0,Y 552.115,Z 289.202,A -85,B 0,C 180,E1 -3448.097,E2 -3448.097} C_VEL
LIN {X 0,Y 552.103,Z 289.213,A -85,B 0,C 180,E1 -3450.627,E2 -3450.627} C_VEL
LIN {X 0,Y 552.119,Z 289.206,A -85,B 0,C 180,E1 -3453.185,E2 -3453.185} C_VEL
LIN {X 0,Y 552.114,Z 289.203,A -85,B 0,C 180,E1 -3453.807,E2 -3453.807} C_VEL
LIN {X 0,Y 551.48,Z 289.288,A -85,B 0,C 180,E1 -3454.415,E2 -3454.415} C_VEL
LIN {X 0,Y 548.654,Z 289.645,A -85,B 0,C 180,E1 -3455.403,E2 -3455.403} C_VEL
LIN {X 0,Y 546.228,Z 289.951,A -85,B 0,C 180,E1 -3456.199,E2 -3456.199} C_VEL
LIN {X 0,Y 545.157,Z 290.081,A -85,B 0,C 180,E1 -3456.813,E2 -3456.813} C_VEL
LIN {X 0,Y 545.055,Z 290.091,A -85,B 0,C 180,E1 -3457.021,E2 -3457.021} C_VEL
LIN {X 0,Y 545.084,Z 290.082,A -85,B 0,C 180,E1 -3460.14,E2 -3460.14} C_VEL
LIN {X 0,Y 545.069,Z 290.087,A -85,B 0,C 180,E1 -3463.107,E2 -3463.107} C_VEL
LIN {X 0,Y 545.056,Z 290.087,A -85,B 0,C 180,E1 -3466.225,E2 -3466.225} C_VEL
LIN {X 0,Y 545.089,Z 290.082,A -85,B 0,C 180,E1 -3468.887,E2 -3468.887} C_VEL
LIN {X 0,Y 545.046,Z 290.087,A -85,B 0,C 180,E1 -3471.763,E2 -3471.763} C_VEL
LIN {X 0,Y 545.058,Z 290.087,A -85,B 0,C 180,E1 -3474.534,E2 -3474.534} C_VEL
LIN {X 0,Y 545.077,Z 290.083,A -85,B 0,C 180,E1 -3477.213,E2 -3477.213} C_VEL
LIN {X 0,Y 545.06,Z 290.086,A -85,B 0,C 180,E1 -3479.811,E2 -3479.811} C_VEL
LIN {X 0,Y 545.091,Z 290.089,A -85,B 0,C 180,E1 -3482.345,E2 -3482.345} C_VEL
LIN {X 0,Y 545.113,Z 290.082,A -85,B 0,C 180,E1 -3484.821,E2 -3484.821} C_VEL
LIN {X 0,Y 545.039,Z 290.089,A -85,B 0,C 180,E1 -3487.243,E2 -3487.243} C_VEL
LIN {X 0,Y 545.116,Z 290.086,A -85,B 0,C 180,E1 -3490.415,E2 -3490.415} C_VEL
LIN {X 0,Y 545.07,Z 290.086,A -85,B 0,C 180,E1 -3493.521,E2 -3493.521} C_VEL
LIN {X 0,Y 545.091,Z 290.086,A -85,B 0,C 180,E1 -3495.82,E2 -3495.82} C_VEL
LIN {X 0,Y 545.115,Z 290.08,A -85,B 0,C 180,E1 -3498.85,E2 -3498.85} C_VEL
LIN {X 0,Y 545.126,Z 290.084,A -85,B 0,C 180,E1 -3501.847,E2 -3501.847} C_VEL
LIN {X 0,Y 545.202,Z 290.069,A -85,B 0,C 180,E1 -3504.823,E2 -3504.823} C_VEL
LIN {X 0,Y 545.196,Z 290.075,A -85,B 0,C 180,E1 -3507.784,E2 -3507.784} C_VEL
LIN {X 0,Y 545.21,Z 290.068,A -85,B 0,C 180,E1 -3510.739,E2 -3510.739} C_VEL
LIN {X 0,Y 545.169,Z 290.073,A -85,B 0,C 180,E1 -3512.956,E2 -3512.956} C_VEL
LIN {X 0,Y 545.171,Z 290.08,A -85,B 0,C 180,E1 -3515.919,E2 -3515.919} C_VEL
LIN {X 0,Y 545.115,Z 290.08,A -85,B 0,C 180,E1 -3518.9,E2 -3518.9} C_VEL
LIN {X 0,Y 545.131,Z 290.085,A -85,B 0,C 180,E1 -3521.904,E2 -3521.904} C_VEL
LIN {X 0,Y 545.082,Z 290.084,A -85,B 0,C 180,E1 -3524.943,E2 -3524.943} C_VEL
LIN {X 0,Y 545.079,Z 290.089,A -85,B 0,C 180,E1 -3528.025,E2 -3528.025} C_VEL
LIN {X 0,Y 545.091,Z 290.083,A -85,B 0,C 180,E1 -3530.372,E2 -3530.372} C_VEL
LIN {X 0,Y 545.086,Z 290.09,A -85,B 0,C 180,E1 -3533.558,E2 -3533.558} C_VEL
LIN {X 0,Y 545.084,Z 290.087,A -85,B 0,C 180,E1 -3536,E2 -3536} C_VEL
LIN {X 0,Y 545.085,Z 290.08,A -85,B 0,C 180,E1 -3538.748,E2 -3538.748} C_VEL
LIN {X 0,Y 545.072,Z 290.091,A -85,B 0,C 180,E1 -3541.682,E2 -3541.682} C_VEL
LIN {X 0,Y 545.077,Z 290.076,A -85,B 0,C 180,E1 -3544.562,E2 -3544.562} C_VEL
LIN {X 0,Y 545.033,Z 290.094,A -85,B 0,C 180,E1 -3547.303,E2 -3547.303} C_VEL
LIN {X 0,Y 545.067,Z 290.081,A -85,B 0,C 180,E1 -3550.141,E2 -3550.141} C_VEL
LIN {X 0,Y 545.078,Z 290.077,A -85,B 0,C 180,E1 -3553.105,E2 -3553.105} C_VEL
LIN {X 0,Y 545.058,Z 290.085,A -85,B 0,C 180,E1 -3556.224,E2 -3556.224} C_VEL
LIN {X 0,Y 545.092,Z 290.082,A -85,B 0,C 180,E1 -3558.887,E2 -3558.887} C_VEL
LIN {X 0,Y 545.045,Z 290.09,A -85,B 0,C 180,E1 -3561.763,E2 -3561.763} C_VEL
LIN {X 0,Y 545.056,Z 290.084,A -85,B 0,C 180,E1 -3564.534,E2 -3564.534} C_VEL
LIN {X 0,Y 545.073,Z 290.09,A -85,B 0,C 180,E1 -3567.212,E2 -3567.212} C_VEL
LIN {X 0,Y 545.092,Z 290.082,A -85,B 0,C 180,E1 -3569.813,E2 -3569.813} C_VEL
LIN {X 0,Y 545.086,Z 290.082,A -85,B 0,C 180,E1 -3572.826,E2 -3572.826} C_VEL
LIN {X 0,Y 545.042,Z 290.089,A -85,B 0,C 180,E1 -3575.631,E2 -3575.631} C_VEL
LIN {X 0,Y 545.059,Z 290.09,A -85,B 0,C 180,E1 -3578.837,E2 -3578.837} C_VEL
LIN {X 0,Y 545.074,Z 290.086,A -85,B 0,C 180,E1 -3581.196,E2 -3581.196} C_VEL
LIN {X 0,Y 545.067,Z 290.086,A -85,B 0,C 180,E1 -3583.521,E2 -3583.521} C_VEL
LIN {X 0,Y 545.085,Z 290.082,A -85,B 0,C 180,E1 -3585.82,E2 -3585.82} C_VEL
LIN {X 0,Y 545.122,Z 290.081,A -85,B 0,C 180,E1 -3588.85,E2 -3588.85} C_VEL
LIN {X 0,Y 545.12,Z 290.074,A -85,B 0,C 180,E1 -3591.847,E2 -3591.847} C_VEL
LIN {X 0,Y 545.198,Z 290.077,A -85,B 0,C 180,E1 -3594.823,E2 -3594.823} C_VEL
LIN {X 0,Y 545.183,Z 290.066,A -85,B 0,C 180,E1 -3597.784,E2 -3597.784} C_VEL
LIN {X 0,Y 545.208,Z 290.067,A -85,B 0,C 180,E1 -3600.739,E2 -3600.739} C_VEL
LIN {X 0,Y 545.166,Z 290.077,A -85,B 0,C 180,E1 -3602.956,E2 -3602.956} C_VEL
LIN {X 0,Y 545.16,Z 290.072,A -85,B 0,C 180,E1 -3605.92,E2 -3605.92} C_VEL
LIN {X 0,Y 545.118,Z 290.075,A -85,B 0,C 180,E1 -3608.9,E2 -3608.9} C_VEL
LIN {X 0,Y 545.127,Z 290.074,A -85,B 0,C 180,E1 -3611.905,E2 -3611.905} C_VEL
LIN {X 0,Y 545.076,Z 290.085,A -85,B 0,C 180,E1 -3614.944,E2 -3614.944} C_VEL
LIN {X 0,Y 545.071,Z 290.081,A -85,B 0,C 180,E1 -3618.026,E2 -3618.026} C_VEL
LIN {X 0,Y 545.091,Z 290.084,A -85,B 0,C 180,E1 -3620.373,E2 -3620.373} C_VEL
LIN {X 0,Y 545.073,Z 290.083,A -85,B 0,C 180,E1 -3623.56,E2 -3623.56} C_VEL
LIN {X 0,Y 545.072,Z 290.084,A -85,B 0,C 180,E1 -3626.001,E2 -3626.001} C_VEL
LIN {X 0,Y 545.083,Z 290.085,A -85,B 0,C 180,E1 -3628.749,E2 -3628.749} C_VEL
LIN {X 0,Y 545.05,Z 290.087,A -85,B 0,C 180,E1 -3631.68,E2 -3631.68} C_VEL
LIN {X 0,Y 545.054,Z 290.089,A -85,B 0,C 180,E1 -3634.565,E2 -3634.565} C_VEL
LIN {X 0,Y 545.03,Z 290.089,A -85,B 0,C 180,E1 -3637.305,E2 -3637.305} C_VEL
LIN {X 0,Y 545.06,Z 290.09,A -85,B 0,C 180,E1 -3640.144,E2 -3640.144} C_VEL
LIN {X 0,Y 545.074,Z 290.083,A -85,B 0,C 180,E1 -3643.107,E2 -3643.107} C_VEL
LIN {X 0,Y 545.046,Z 290.095,A -85,B 0,C 180,E1 -3646.227,E2 -3646.227} C_VEL
LIN {X 0,Y 545.077,Z 290.078,A -85,B 0,C 180,E1 -3648.886,E2 -3648.886} C_VEL
LIN {X 0,Y 545.076,Z 290.083,A -85,B 0,C 180,E1 -3650.819,E2 -3650.819} C_VEL
LIN {X 0,Y 545.032,Z 290.091,A -85,B 0,C 180,E1 -3653.62,E2 -3653.62} C_VEL
LIN {X 0,Y 545.064,Z 290.089,A -85,B 0,C 180,E1 -3656.329,E2 -3656.329} C_VEL
LIN {X 0,Y 545.065,Z 290.086,A -85,B 0,C 180,E1 -3658.953,E2 -3658.953} C_VEL
LIN {X 0,Y 545.082,Z 290.088,A -85,B 0,C 180,E1 -3661.507,E2 -3661.507} C_VEL
LIN {X 0,Y 545.117,Z 290.204,A -85,B 0,C 180,E1 -3664.487,E2 -3664.487} C_VEL
LIN {X 0,Y 546.05,Z 295.944,A -85,B 0,C 180,E1 -3665.679,E2 -3665.679} C_VEL
LIN {X 0,Y 545.72,Z 311.498,A -85,B 0,C 180,E1 -3668.666,E2 -3668.666} C_VEL
LIN {X 0,Y 545.488,Z 328.233,A -85,B 0,C 180,E1 -3671.794,E2 -3671.794} C_VEL
LIN {X 0,Y 545.239,Z 344.935,A -85,B 0,C 180,E1 -3674.87,E2 -3674.87} C_VEL
LIN {X 0,Y 545.18,Z 348.282,A -85,B 0,C 180,E1 -3675.434,E2 -3675.434} C_VEL
LIN {X 0,Y 546.547,Z 357.582,A -85,B 0,C 180,E1 -3675.619,E2 -3675.619} C_VEL
LIN {X 0,Y 546.242,Z 453.069,A -85,B 0,C 180,E1 -3676.894,E2 -3676.894} C_VEL
LIN {X 0,Y 546.135,Z 462.962,A -85,B 0,C 180,E1 -3677.104,E2 -3677.104} C_VEL
LIN {X 0,Y 546.013,Z 472.938,A -85,B 0,C 180,E1 -3677.408,E2 -3677.408} C_VEL
LIN {X 0,Y 545.853,Z 482.296,A -85,B 0,C 180,E1 -3677.782,E2 -3677.782} C_VEL
LIN {X 0,Y 545.685,Z 492.48,A -85,B 0,C 180,E1 -3678.299,E2 -3678.299} C_VEL
LIN {X 0,Y 545.549,Z 501.441,A -85,B 0,C 180,E1 -3678.859,E2 -3678.859} C_VEL
LIN {X 0,Y 545.392,Z 510.148,A -85,B 0,C 180,E1 -3679.513,E2 -3679.513} C_VEL
LIN {X 0,Y 545.221,Z 517.519,A -85,B 0,C 180,E1 -3680.166,E2 -3680.166} C_VEL
LIN {X 0,Y 545.099,Z 524.713,A -85,B 0,C 180,E1 -3680.913,E2 -3680.913} C_VEL
LIN {X 0,Y 544.973,Z 530.889,A -85,B 0,C 180,E1 -3681.658,E2 -3681.658} C_VEL
LIN {X 0,Y 544.836,Z 537.397,A -85,B 0,C 180,E1 -3682.589,E2 -3682.589} C_VEL
LIN {X 0,Y 544.76,Z 542.262,A -85,B 0,C 180,E1 -3683.408,E2 -3683.408} C_VEL
LIN {X 0,Y 544.738,Z 547.335,A -85,B 0,C 180,E1 -3684.447,E2 -3684.447} C_VEL
LIN {X 0,Y 544.664,Z 551.63,A -85,B 0,C 180,E1 -3685.56,E2 -3685.56} C_VEL
LIN {X 0,Y 544.669,Z 553.974,A -85,B 0,C 180,E1 -3686.301,E2 -3686.301} C_VEL
LIN {X 0,Y 544.65,Z 555.762,A -85,B 0,C 180,E1 -3687.041,E2 -3687.041} C_VEL
LIN {X 0,Y 544.546,Z 558.189,A -85,B 0,C 180,E1 -3688.521,E2 -3688.521} C_VEL
LIN {X 0,Y 544.542,Z 558.772,A -85,B 0,C 180,E1 -3689.261,E2 -3689.261} C_VEL
LIN {X 0,Y 544.542,Z 558.772,A -85,B 0,C 180,E1 -3690.739,E2 -3690.739} C_VEL
LIN {X 0,Y 544.546,Z 558.189,A -85,B 0,C 180,E1 -3691.479,E2 -3691.479} C_VEL
LIN {X 0,Y 544.65,Z 555.762,A -85,B 0,C 180,E1 -3692.959,E2 -3692.959} C_VEL
LIN {X 0,Y 544.684,Z 552.838,A -85,B 0,C 180,E1 -3694.069,E2 -3694.069} C_VEL
LIN {X 0,Y 544.653,Z 548.879,A -85,B 0,C 180,E1 -3695.182,E2 -3695.182} C_VEL
LIN {X 0,Y 544.759,Z 544.638,A -85,B 0,C 180,E1 -3696.128,E2 -3696.128} C_VEL
LIN {X 0,Y 544.79,Z 539.697,A -85,B 0,C 180,E1 -3697.039,E2 -3697.039} C_VEL
LIN {X 0,Y 544.916,Z 533.63,A -85,B 0,C 180,E1 -3697.969,E2 -3697.969} C_VEL
LIN {X 0,Y 545.038,Z 526.333,A -85,B 0,C 180,E1 -3698.901,E2 -3698.901} C_VEL
LIN {X 0,Y 545.198,Z 519.432,A -85,B 0,C 180,E1 -3699.647,E2 -3699.647} C_VEL
LIN {X 0,Y 545.349,Z 511.279,A -85,B 0,C 180,E1 -3700.394,E2 -3700.394} C_VEL
LIN {X 0,Y 545.525,Z 502.791,A -85,B 0,C 180,E1 -3701.048,E2 -3701.048} C_VEL
LIN {X 0,Y 545.699,Z 493.465,A -85,B 0,C 180,E1 -3701.644,E2 -3701.644} C_VEL
LIN {X 0,Y 545.84,Z 483.304,A -85,B 0,C 180,E1 -3702.171,E2 -3702.171} C_VEL
LIN {X 0,Y 545.986,Z 474.226,A -85,B 0,C 180,E1 -3702.545,E2 -3702.545} C_VEL
LIN {X 0,Y 546.128,Z 464.711,A -85,B 0,C 180,E1 -3702.849,E2 -3702.849} C_VEL
LIN {X 0,Y 546.208,Z 454.4,A -85,B 0,C 180,E1 -3703.084,E2 -3703.084} C_VEL
LIN {X 0,Y 546.417,Z 398.906,A -85,B 0,C 180,E1 -3703.836,E2 -3703.836} C_VEL
LIN {X 0,Y 546.401,Z 355.337,A -85,B 0,C 180,E1 -3704.415,E2 -3704.415} C_VEL
LIN {X 0,Y 545.18,Z 348.279,A -85,B 0,C 180,E1 -3704.566,E2 -3704.566} C_VEL
LIN {X 0,Y 545.303,Z 338.676,A -85,B 0,C 180,E1 -3706.279,E2 -3706.279} C_VEL
LIN {X 0,Y 545.489,Z 324.051,A -85,B 0,C 180,E1 -3708.984,E2 -3708.984} C_VEL
LIN {X 0,Y 545.776,Z 309.467,A -85,B 0,C 180,E1 -3711.728,E2 -3711.728} C_VEL
LIN {X 0,Y 546.046,Z 295.97,A -85,B 0,C 180,E1 -3714.321,E2 -3714.321} C_VEL
LIN {X 0,Y 545.092,Z 290.115,A -85,B 0,C 180,E1 -3715.555,E2 -3715.555} C_VEL
LIN {X 0,Y 545.082,Z 290.088,A -85,B 0,C 180,E1 -3718.493,E2 -3718.493} C_VEL
LIN {X 0,Y 545.065,Z 290.086,A -85,B 0,C 180,E1 -3721.047,E2 -3721.047} C_VEL
LIN {X 0,Y 545.064,Z 290.089,A -85,B 0,C 180,E1 -3723.671,E2 -3723.671} C_VEL
LIN {X 0,Y 545.063,Z 290.084,A -85,B 0,C 180,E1 -3726.924,E2 -3726.924} C_VEL
LIN {X 0,Y 545.062,Z 290.085,A -85,B 0,C 180,E1 -3730.142,E2 -3730.142} C_VEL
LIN {X 0,Y 545.075,Z 290.084,A -85,B 0,C 180,E1 -3733.106,E2 -3733.106} C_VEL
LIN {X 0,Y 545.046,Z 290.09,A -85,B 0,C 180,E1 -3736.225,E2 -3736.225} C_VEL
LIN {X 0,Y 545.091,Z 290.08,A -85,B 0,C 180,E1 -3738.886,E2 -3738.886} C_VEL
LIN {X 0,Y 545.047,Z 290.095,A -85,B 0,C 180,E1 -3741.762,E2 -3741.762} C_VEL
LIN {X 0,Y 545.031,Z 290.087,A -85,B 0,C 180,E1 -3744.531,E2 -3744.531} C_VEL
LIN {X 0,Y 545.059,Z 290.085,A -85,B 0,C 180,E1 -3747.21,E2 -3747.21} C_VEL
LIN {X 0,Y 545.056,Z 290.091,A -85,B 0,C 180,E1 -3749.81,E2 -3749.81} C_VEL
LIN {X 0,Y 545.086,Z 290.078,A -85,B 0,C 180,E1 -3752.344,E2 -3752.344} C_VEL
LIN {X 0,Y 545.109,Z 290.076,A -85,B 0,C 180,E1 -3754.82,E2 -3754.82} C_VEL
LIN {X 0,Y 545.03,Z 290.093,A -85,B 0,C 180,E1 -3757.242,E2 -3757.242} C_VEL
LIN {X 0,Y 545.113,Z 290.073,A -85,B 0,C 180,E1 -3760.414,E2 -3760.414} C_VEL
LIN {X 0,Y 545.067,Z 290.09,A -85,B 0,C 180,E1 -3763.521,E2 -3763.521} C_VEL
LIN {X 0,Y 545.087,Z 290.084,A -85,B 0,C 180,E1 -3765.819,E2 -3765.819} C_VEL
LIN {X 0,Y 545.122,Z 290.076,A -85,B 0,C 180,E1 -3768.849,E2 -3768.849} C_VEL
LIN {X 0,Y 545.125,Z 290.076,A -85,B 0,C 180,E1 -3771.847,E2 -3771.847} C_VEL
LIN {X 0,Y 545.198,Z 290.07,A -85,B 0,C 180,E1 -3774.822,E2 -3774.822} C_VEL
LIN {X 0,Y 545.182,Z 290.069,A -85,B 0,C 180,E1 -3777.783,E2 -3777.783} C_VEL
LIN {X 0,Y 545.207,Z 290.061,A -85,B 0,C 180,E1 -3780.738,E2 -3780.738} C_VEL
LIN {X 0,Y 545.168,Z 290.074,A -85,B 0,C 180,E1 -3782.955,E2 -3782.955} C_VEL
LIN {X 0,Y 545.16,Z 290.072,A -85,B 0,C 180,E1 -3785.919,E2 -3785.919} C_VEL
LIN {X 0,Y 545.112,Z 290.081,A -85,B 0,C 180,E1 -3788.9,E2 -3788.9} C_VEL
LIN {X 0,Y 545.125,Z 290.074,A -85,B 0,C 180,E1 -3791.904,E2 -3791.904} C_VEL
LIN {X 0,Y 545.075,Z 290.091,A -85,B 0,C 180,E1 -3794.943,E2 -3794.943} C_VEL
LIN {X 0,Y 545.068,Z 290.08,A -85,B 0,C 180,E1 -3798.026,E2 -3798.026} C_VEL
LIN {X 0,Y 545.088,Z 290.078,A -85,B 0,C 180,E1 -3800.372,E2 -3800.372} C_VEL
LIN {X 0,Y 545.081,Z 290.083,A -85,B 0,C 180,E1 -3803.559,E2 -3803.559} C_VEL
LIN {X 0,Y 545.069,Z 290.081,A -85,B 0,C 180,E1 -3806.001,E2 -3806.001} C_VEL
LIN {X 0,Y 545.083,Z 290.086,A -85,B 0,C 180,E1 -3808.749,E2 -3808.749} C_VEL
LIN {X 0,Y 545.068,Z 290.084,A -85,B 0,C 180,E1 -3811.683,E2 -3811.683} C_VEL
LIN {X 0,Y 545.075,Z 290.087,A -85,B 0,C 180,E1 -3814.563,E2 -3814.563} C_VEL
LIN {X 0,Y 545.055,Z 290.091,A -85,B 0,C 180,E1 -3817.021,E2 -3817.021} C_VEL
LIN {X 0,Y 544.35,Z 290.176,A -85,B 0,C 180,E1 -3817.637,E2 -3817.637} C_VEL
LIN {X 0,Y 541.496,Z 290.538,A -85,B 0,C 180,E1 -3818.638,E2 -3818.638} C_VEL
LIN {X 0,Y 539.119,Z 290.828,A -85,B 0,C 180,E1 -3819.444,E2 -3819.444} C_VEL
LIN {X 0,Y 538.114,Z 290.95,A -85,B 0,C 180,E1 -3820.066,E2 -3820.066} C_VEL
LIN {X 0,Y 538.039,Z 290.959,A -85,B 0,C 180,E1 -3820.277,E2 -3820.277} C_VEL
LIN {X 0,Y 538.017,Z 290.967,A -85,B 0,C 180,E1 -3822.988,E2 -3822.988} C_VEL
LIN {X 0,Y 538.02,Z 290.96,A -85,B 0,C 180,E1 -3825.926,E2 -3825.926} C_VEL
LIN {X 0,Y 538.044,Z 290.956,A -85,B 0,C 180,E1 -3829.225,E2 -3829.225} C_VEL
LIN {X 0,Y 537.987,Z 290.97,A -85,B 0,C 180,E1 -3832.123,E2 -3832.123} C_VEL
LIN {X 0,Y 538.014,Z 290.958,A -85,B 0,C 180,E1 -3834.918,E2 -3834.918} C_VEL
LIN {X 0,Y 538.026,Z 290.961,A -85,B 0,C 180,E1 -3837.619,E2 -3837.619} C_VEL
LIN {X 0,Y 538.013,Z 290.967,A -85,B 0,C 180,E1 -3840.239,E2 -3840.239} C_VEL
LIN {X 0,Y 538.066,Z 290.96,A -85,B 0,C 180,E1 -3842.797,E2 -3842.797} C_VEL
LIN {X 0,Y 538.044,Z 290.96,A -85,B 0,C 180,E1 -3845.293,E2 -3845.293} C_VEL
LIN {X 0,Y 538.01,Z 290.97,A -85,B 0,C 180,E1 -3848.042,E2 -3848.042} C_VEL
LIN {X 0,Y 538.036,Z 290.962,A -85,B 0,C 180,E1 -3850.94,E2 -3850.94} C_VEL
LIN {X 0,Y 538.021,Z 290.963,A -85,B 0,C 180,E1 -3853.299,E2 -3853.299} C_VEL
LIN {X 0,Y 538.06,Z 290.96,A -85,B 0,C 180,E1 -3855.631,E2 -3855.631} C_VEL
LIN {X 0,Y 538.074,Z 290.959,A -85,B 0,C 180,E1 -3858.702,E2 -3858.702} C_VEL
LIN {X 0,Y 538.083,Z 290.96,A -85,B 0,C 180,E1 -3861.74,E2 -3861.74} C_VEL
LIN {X 0,Y 538.16,Z 290.947,A -85,B 0,C 180,E1 -3864.755,E2 -3864.755} C_VEL
LIN {X 0,Y 538.167,Z 290.951,A -85,B 0,C 180,E1 -3867.755,E2 -3867.755} C_VEL
LIN {X 0,Y 538.18,Z 290.944,A -85,B 0,C 180,E1 -3870.748,E2 -3870.748} C_VEL
LIN {X 0,Y 538.136,Z 290.949,A -85,B 0,C 180,E1 -3872.994,E2 -3872.994} C_VEL
LIN {X 0,Y 538.123,Z 290.958,A -85,B 0,C 180,E1 -3875.997,E2 -3875.997} C_VEL
LIN {X 0,Y 538.066,Z 290.958,A -85,B 0,C 180,E1 -3879.017,E2 -3879.017} C_VEL
LIN {X 0,Y 538.08,Z 290.962,A -85,B 0,C 180,E1 -3882.062,E2 -3882.062} C_VEL
LIN {X 0,Y 538.041,Z 290.962,A -85,B 0,C 180,E1 -3885.143,E2 -3885.143} C_VEL
LIN {X 0,Y 538.031,Z 290.964,A -85,B 0,C 180,E1 -3888.27,E2 -3888.27} C_VEL
LIN {X 0,Y 538.035,Z 290.961,A -85,B 0,C 180,E1 -3890.651,E2 -3890.651} C_VEL
LIN {X 0,Y 538.019,Z 290.969,A -85,B 0,C 180,E1 -3893.887,E2 -3893.887} C_VEL
LIN {X 0,Y 538.045,Z 290.96,A -85,B 0,C 180,E1 -3896.366,E2 -3896.366} C_VEL
LIN {X 0,Y 538.026,Z 290.96,A -85,B 0,C 180,E1 -3898.933,E2 -3898.933} C_VEL
LIN {X 0,Y 538.022,Z 290.966,A -85,B 0,C 180,E1 -3901.89,E2 -3901.89} C_VEL
LIN {X 0,Y 538.027,Z 290.954,A -85,B 0,C 180,E1 -3904.621,E2 -3904.621} C_VEL
LIN {X 0,Y 538.001,Z 290.968,A -85,B 0,C 180,E1 -3907.17,E2 -3907.17} C_VEL
LIN {X 0,Y 538.022,Z 290.962,A -85,B 0,C 180,E1 -3909.796,E2 -3909.796} C_VEL
LIN {X 0,Y 538.015,Z 290.953,A -85,B 0,C 180,E1 -3912.785,E2 -3912.785} C_VEL
LIN {X 0,Y 538.021,Z 290.964,A -85,B 0,C 180,E1 -3915.925,E2 -3915.925} C_VEL
LIN {X 0,Y 538.069,Z 290.961,A -85,B 0,C 180,E1 -3919.249,E2 -3919.249} C_VEL
LIN {X 0,Y 537.985,Z 290.967,A -85,B 0,C 180,E1 -3922.122,E2 -3922.122} C_VEL
LIN {X 0,Y 538.012,Z 290.965,A -85,B 0,C 180,E1 -3924.917,E2 -3924.917} C_VEL
LIN {X 0,Y 538.022,Z 290.965,A -85,B 0,C 180,E1 -3927.618,E2 -3927.618} C_VEL
LIN {X 0,Y 538.033,Z 290.96,A -85,B 0,C 180,E1 -3930.24,E2 -3930.24} C_VEL
LIN {X 0,Y 538.056,Z 290.956,A -85,B 0,C 180,E1 -3932.796,E2 -3932.796} C_VEL
LIN {X 0,Y 538.039,Z 290.966,A -85,B 0,C 180,E1 -3935.293,E2 -3935.293} C_VEL
LIN {X 0,Y 538.004,Z 290.963,A -85,B 0,C 180,E1 -3938.042,E2 -3938.042} C_VEL
LIN {X 0,Y 538.03,Z 290.961,A -85,B 0,C 180,E1 -3940.94,E2 -3940.94} C_VEL
LIN {X 0,Y 538.018,Z 290.966,A -85,B 0,C 180,E1 -3943.299,E2 -3943.299} C_VEL
LIN {X 0,Y 538.053,Z 290.959,A -85,B 0,C 180,E1 -3945.631,E2 -3945.631} C_VEL
LIN {X 0,Y 538.079,Z 290.957,A -85,B 0,C 180,E1 -3948.702,E2 -3948.702} C_VEL
LIN {X 0,Y 538.077,Z 290.951,A -85,B 0,C 180,E1 -3951.74,E2 -3951.74} C_VEL
LIN {X 0,Y 538.154,Z 290.953,A -85,B 0,C 180,E1 -3954.755,E2 -3954.755} C_VEL
LIN {X 0,Y 538.155,Z 290.941,A -85,B 0,C 180,E1 -3957.755,E2 -3957.755} C_VEL
LIN {X 0,Y 538.178,Z 290.942,A -85,B 0,C 180,E1 -3960.749,E2 -3960.749} C_VEL
LIN {X 0,Y 538.132,Z 290.953,A -85,B 0,C 180,E1 -3962.995,E2 -3962.995} C_VEL
LIN {X 0,Y 538.113,Z 290.951,A -85,B 0,C 180,E1 -3965.998,E2 -3965.998} C_VEL
LIN {X 0,Y 538.067,Z 290.951,A -85,B 0,C 180,E1 -3969.018,E2 -3969.018} C_VEL
LIN {X 0,Y 538.075,Z 290.954,A -85,B 0,C 180,E1 -3972.063,E2 -3972.063} C_VEL
LIN {X 0,Y 538.036,Z 290.96,A -85,B 0,C 180,E1 -3975.144,E2 -3975.144} C_VEL
LIN {X 0,Y 538.024,Z 290.961,A -85,B 0,C 180,E1 -3978.271,E2 -3978.271} C_VEL
LIN {X 0,Y 538.034,Z 290.966,A -85,B 0,C 180,E1 -3980.652,E2 -3980.652} C_VEL
LIN {X 0,Y 537.996,Z 290.966,A -85,B 0,C 180,E1 -3983.889,E2 -3983.889} C_VEL
LIN {X 0,Y 538.035,Z 290.963,A -85,B 0,C 180,E1 -3986.367,E2 -3986.367} C_VEL
LIN {X 0,Y 538.024,Z 290.963,A -85,B 0,C 180,E1 -3988.934,E2 -3988.934} C_VEL
LIN {X 0,Y 538.003,Z 290.967,A -85,B 0,C 180,E1 -3991.888,E2 -3991.888} C_VEL
LIN {X 0,Y 538.004,Z 290.966,A -85,B 0,C 180,E1 -3994.618,E2 -3994.618} C_VEL
LIN {X 0,Y 537.998,Z 290.965,A -85,B 0,C 180,E1 -3997.171,E2 -3997.171} C_VEL
LIN {X 0,Y 538.017,Z 290.963,A -85,B 0,C 180,E1 -3999.798,E2 -3999.798} C_VEL
LIN {X 0,Y 538.015,Z 290.964,A -85,B 0,C 180,E1 -4002.787,E2 -4002.787} C_VEL
LIN {X 0,Y 538.016,Z 290.968,A -85,B 0,C 180,E1 -4005.927,E2 -4005.927} C_VEL
LIN {X 0,Y 538.045,Z 290.953,A -85,B 0,C 180,E1 -4009.225,E2 -4009.225} C_VEL
LIN {X 0,Y 537.986,Z 290.974,A -85,B 0,C 180,E1 -4012.123,E2 -4012.123} C_VEL
LIN {X 0,Y 537.993,Z 290.965,A -85,B 0,C 180,E1 -4014.916,E2 -4014.916} C_VEL
LIN {X 0,Y 538.017,Z 290.966,A -85,B 0,C 180,E1 -4017.618,E2 -4017.618} C_VEL
LIN {X 0,Y 538.013,Z 290.969,A -85,B 0,C 180,E1 -4020.239,E2 -4020.239} C_VEL
LIN {X 0,Y 538.048,Z 290.963,A -85,B 0,C 180,E1 -4022.796,E2 -4022.796} C_VEL
LIN {X 0,Y 538.084,Z 291.075,A -85,B 0,C 180,E1 -4024.319,E2 -4024.319} C_VEL
LIN {X 0,Y 539.106,Z 297.456,A -85,B 0,C 180,E1 -4025.662,E2 -4025.662} C_VEL
LIN {X 0,Y 538.75,Z 312.423,A -85,B 0,C 180,E1 -4028.577,E2 -4028.577} C_VEL
LIN {X 0,Y 538.466,Z 329.144,A -85,B 0,C 180,E1 -4031.746,E2 -4031.746} C_VEL
LIN {X 0,Y 538.196,Z 345.8,A -85,B 0,C 180,E1 -4034.861,E2 -4034.861} C_VEL
LIN {X 0,Y 538.137,Z 348.086,A -85,B 0,C 180,E1 -4035.24,E2 -4035.24} C_VEL
LIN {X 0,Y 539.677,Z 358.023,A -85,B 0,C 180,E1 -4035.441,E2 -4035.441} C_VEL
LIN {X 0,Y 539.332,Z 452.875,A -85,B 0,C 180,E1 -4036.723,E2 -4036.723} C_VEL
LIN {X 0,Y 539.192,Z 462.767,A -85,B 0,C 180,E1 -4036.935,E2 -4036.935} C_VEL
LIN {X 0,Y 539.093,Z 472.745,A -85,B 0,C 180,E1 -4037.244,E2 -4037.244} C_VEL
LIN {X 0,Y 538.898,Z 482.102,A -85,B 0,C 180,E1 -4037.622,E2 -4037.622} C_VEL
LIN {X 0,Y 538.739,Z 492.047,A -85,B 0,C 180,E1 -4038.132,E2 -4038.132} C_VEL
LIN {X 0,Y 538.549,Z 501.247,A -85,B 0,C 180,E1 -4038.712,E2 -4038.712} C_VEL
LIN {X 0,Y 538.366,Z 509.978,A -85,B 0,C 180,E1 -4039.375,E2 -4039.375} C_VEL
LIN {X 0,Y 538.189,Z 517.375,A -85,B 0,C 180,E1 -4040.036,E2 -4040.036} C_VEL
LIN {X 0,Y 538.055,Z 524.597,A -85,B 0,C 180,E1 -4040.793,E2 -4040.793} C_VEL
LIN {X 0,Y 537.913,Z 530.799,A -85,B 0,C 180,E1 -4041.548,E2 -4041.548} C_VEL
LIN {X 0,Y 537.772,Z 537.335,A -85,B 0,C 180,E1 -4042.491,E2 -4042.491} C_VEL
LIN {X 0,Y 537.673,Z 542.724,A -85,B 0,C 180,E1 -4043.419,E2 -4043.419} C_VEL
LIN {X 0,Y 537.673,Z 547.323,A -85,B 0,C 180,E1 -4044.374,E2 -4044.374} C_VEL
LIN {X 0,Y 537.562,Z 551.622,A -85,B 0,C 180,E1 -4045.501,E2 -4045.501} C_VEL
LIN {X 0,Y 537.591,Z 553.972,A -85,B 0,C 180,E1 -4046.252,E2 -4046.252} C_VEL
LIN {X 0,Y 537.551,Z 555.756,A -85,B 0,C 180,E1 -4047.002,E2 -4047.002} C_VEL
LIN {X 0,Y 537.452,Z 558.181,A -85,B 0,C 180,E1 -4048.501,E2 -4048.501} C_VEL
LIN {X 0,Y 537.442,Z 558.764,A -85,B 0,C 180,E1 -4049.251,E2 -4049.251} C_VEL
LIN {X 0,Y 537.442,Z 558.764,A -85,B 0,C 180,E1 -4050.749,E2 -4050.749} C_VEL
LIN {X 0,Y 537.452,Z 558.181,A -85,B 0,C 180,E1 -4051.499,E2 -4051.499} C_VEL
LIN {X 0,Y 537.551,Z 555.756,A -85,B 0,C 180,E1 -4052.998,E2 -4052.998} C_VEL
LIN {X 0,Y 537.604,Z 552.831,A -85,B 0,C 180,E1 -4054.123,E2 -4054.123} C_VEL
LIN {X 0,Y 537.587,Z 548.87,A -85,B 0,C 180,E1 -4055.251,E2 -4055.251} C_VEL
LIN {X 0,Y 537.636,Z 544.059,A -85,B 0,C 180,E1 -4056.318,E2 -4056.318} C_VEL
LIN {X 0,Y 537.754,Z 538.49,A -85,B 0,C 180,E1 -4057.321,E2 -4057.321} C_VEL
LIN {X 0,Y 537.88,Z 532.175,A -85,B 0,C 180,E1 -4058.263,E2 -4058.263} C_VEL
LIN {X 0,Y 537.991,Z 526.223,A -85,B 0,C 180,E1 -4059.019,E2 -4059.019} C_VEL
LIN {X 0,Y 538.15,Z 519.295,A -85,B 0,C 180,E1 -4059.774,E2 -4059.774} C_VEL
LIN {X 0,Y 538.355,Z 511.114,A -85,B 0,C 180,E1 -4060.531,E2 -4060.531} C_VEL
LIN {X 0,Y 538.52,Z 502.599,A -85,B 0,C 180,E1 -4061.193,E2 -4061.193} C_VEL
LIN {X 0,Y 538.711,Z 494.241,A -85,B 0,C 180,E1 -4061.74,E2 -4061.74} C_VEL
LIN {X 0,Y 538.877,Z 484.117,A -85,B 0,C 180,E1 -4062.283,E2 -4062.283} C_VEL
LIN {X 0,Y 539.031,Z 475.321,A -85,B 0,C 180,E1 -4062.662,E2 -4062.662} C_VEL
LIN {X 0,Y 539.192,Z 465.392,A -85,B 0,C 180,E1 -4062.993,E2 -4062.993} C_VEL
LIN {X 0,Y 539.299,Z 455.538,A -85,B 0,C 180,E1 -4063.23,E2 -4063.23} C_VEL
LIN {X 0,Y 539.442,Z 432.723,A -85,B 0,C 180,E1 -4063.562,E2 -4063.562} C_VEL
LIN {X 0,Y 539.635,Z 356.861,A -85,B 0,C 180,E1 -4064.576,E2 -4064.576} C_VEL
LIN {X 0,Y 538.137,Z 348.082,A -85,B 0,C 180,E1 -4064.76,E2 -4064.76} C_VEL
LIN {X 0,Y 538.175,Z 344.797,A -85,B 0,C 180,E1 -4065.334,E2 -4065.334} C_VEL
LIN {X 0,Y 538.466,Z 329.144,A -85,B 0,C 180,E1 -4068.254,E2 -4068.254} C_VEL
LIN {X 0,Y 538.75,Z 312.431,A -85,B 0,C 180,E1 -4071.423,E2 -4071.423} C_VEL
LIN {X 0,Y 539.08,Z 297.492,A -85,B 0,C 180,E1 -4074.338,E2 -4074.338} C_VEL
LIN {X 0,Y 538.054,Z 290.995,A -85,B 0,C 180,E1 -4075.722,E2 -4075.722} C_VEL
LIN {X 0,Y 538.025,Z 290.968,A -85,B 0,C 180,E1 -4078.05,E2 -4078.05} C_VEL
LIN {X 0,Y 538.02,Z 290.966,A -85,B 0,C 180,E1 -4080.626,E2 -4080.626} C_VEL
LIN {X 0,Y 538.045,Z 290.959,A -85,B 0,C 180,E1 -4083.282,E2 -4083.282} C_VEL
LIN {X 0,Y 537.987,Z 290.971,A -85,B 0,C 180,E1 -4086.004,E2 -4086.004} C_VEL
LIN {X 0,Y 538.008,Z 290.963,A -85,B 0,C 180,E1 -4088.83,E2 -4088.83} C_VEL
LIN {X 0,Y 538.026,Z 290.963,A -85,B 0,C 180,E1 -4091.772,E2 -4091.772} C_VEL
LIN {X 0,Y 538.003,Z 290.963,A -85,B 0,C 180,E1 -4094.861,E2 -4094.861} C_VEL
LIN {X 0,Y 538.033,Z 290.964,A -85,B 0,C 180,E1 -4098.12,E2 -4098.12} C_VEL
LIN {X 0,Y 538.03,Z 290.96,A -85,B 0,C 180,E1 -4100.414,E2 -4100.414} C_VEL
LIN {X 0,Y 538.018,Z 290.963,A -85,B 0,C 180,E1 -4103.066,E2 -4103.066} C_VEL
LIN {X 0,Y 538.006,Z 290.967,A -85,B 0,C 180,E1 -4105.825,E2 -4105.825} C_VEL
LIN {X 0,Y 538.001,Z 290.964,A -85,B 0,C 180,E1 -4108.498,E2 -4108.498} C_VEL
LIN {X 0,Y 538.053,Z 290.959,A -85,B 0,C 180,E1 -4111.099,E2 -4111.099} C_VEL
LIN {X 0,Y 538.035,Z 290.963,A -85,B 0,C 180,E1 -4113.633,E2 -4113.633} C_VEL
LIN {X 0,Y 537.999,Z 290.966,A -85,B 0,C 180,E1 -4116.121,E2 -4116.121} C_VEL
LIN {X 0,Y 538.034,Z 290.966,A -85,B 0,C 180,E1 -4119.348,E2 -4119.348} C_VEL
LIN {X 0,Y 538.045,Z 290.953,A -85,B 0,C 180,E1 -4122.516,E2 -4122.516} C_VEL
LIN {X 0,Y 538.055,Z 290.963,A -85,B 0,C 180,E1 -4125.63,E2 -4125.63} C_VEL
LIN {X 0,Y 538.08,Z 290.952,A -85,B 0,C 180,E1 -4128.701,E2 -4128.701} C_VEL
LIN {X 0,Y 538.081,Z 290.954,A -85,B 0,C 180,E1 -4131.739,E2 -4131.739} C_VEL
LIN {X 0,Y 538.155,Z 290.947,A -85,B 0,C 180,E1 -4134.755,E2 -4134.755} C_VEL
LIN {X 0,Y 538.154,Z 290.944,A -85,B 0,C 180,E1 -4137.754,E2 -4137.754} C_VEL
LIN {X 0,Y 538.177,Z 290.936,A -85,B 0,C 180,E1 -4140.748,E2 -4140.748} C_VEL
LIN {X 0,Y 538.134,Z 290.95,A -85,B 0,C 180,E1 -4142.994,E2 -4142.994} C_VEL
LIN {X 0,Y 538.113,Z 290.95,A -85,B 0,C 180,E1 -4145.997,E2 -4145.997} C_VEL
LIN {X 0,Y 538.062,Z 290.959,A -85,B 0,C 180,E1 -4149.017,E2 -4149.017} C_VEL
LIN {X 0,Y 538.073,Z 290.952,A -85,B 0,C 180,E1 -4152.062,E2 -4152.062} C_VEL
LIN {X 0,Y 538.035,Z 290.967,A -85,B 0,C 180,E1 -4155.144,E2 -4155.144} C_VEL
LIN {X 0,Y 538.021,Z 290.958,A -85,B 0,C 180,E1 -4158.27,E2 -4158.27} C_VEL
LIN {X 0,Y 538.032,Z 290.96,A -85,B 0,C 180,E1 -4160.651,E2 -4160.651} C_VEL
LIN {X 0,Y 538.013,Z 290.963,A -85,B 0,C 180,E1 -4163.887,E2 -4163.887} C_VEL
LIN {X 0,Y 538.032,Z 290.96,A -85,B 0,C 180,E1 -4166.367,E2 -4166.367} C_VEL
LIN {X 0,Y 538.046,Z 290.966,A -85,B 0,C 180,E1 -4168.939,E2 -4168.939} C_VEL
LIN {X 0,Y 538.017,Z 290.962,A -85,B 0,C 180,E1 -4171.89,E2 -4171.89} C_VEL
LIN {X 0,Y 538.025,Z 290.965,A -85,B 0,C 180,E1 -4174.622,E2 -4174.622} C_VEL
LIN {X 0,Y 537.998,Z 290.968,A -85,B 0,C 180,E1 -4177.171,E2 -4177.171} C_VEL
LIN {X 0,Y 538.039,Z 290.959,A -85,B 0,C 180,E1 -4180.277,E2 -4180.277} C_VEL
LIN {X 0,Y 537.387,Z 291.045,A -85,B 0,C 180,E1 -4180.902,E2 -4180.902} C_VEL
LIN {X 0,Y 534.526,Z 291.401,A -85,B 0,C 180,E1 -4181.916,E2 -4181.916} C_VEL
LIN {X 0,Y 532.092,Z 291.709,A -85,B 0,C 180,E1 -4182.733,E2 -4182.733} C_VEL
LIN {X 0,Y 531.041,Z 291.833,A -85,B 0,C 180,E1 -4183.364,E2 -4183.364} C_VEL
LIN {X 0,Y 530.953,Z 291.842,A -85,B 0,C 180,E1 -4183.578,E2 -4183.578} C_VEL
LIN {X 0,Y 530.958,Z 291.841,A -85,B 0,C 180,E1 -4186.506,E2 -4186.506} C_VEL
LIN {X 0,Y 530.982,Z 291.837,A -85,B 0,C 180,E1 -4188.976,E2 -4188.976} C_VEL
LIN {X 0,Y 530.952,Z 291.843,A -85,B 0,C 180,E1 -4191.53,E2 -4191.53} C_VEL
LIN {X 0,Y 530.975,Z 291.842,A -85,B 0,C 180,E1 -4194.383,E2 -4194.383} C_VEL
LIN {X 0,Y 530.969,Z 291.841,A -85,B 0,C 180,E1 -4197.134,E2 -4197.134} C_VEL
LIN {X 0,Y 530.964,Z 291.842,A -85,B 0,C 180,E1 -4199.803,E2 -4199.803} C_VEL
LIN {X 0,Y 531.012,Z 291.844,A -85,B 0,C 180,E1 -4202.467,E2 -4202.467} C_VEL
LIN {X 0,Y 531.003,Z 291.839,A -85,B 0,C 180,E1 -4204.943,E2 -4204.943} C_VEL
LIN {X 0,Y 530.967,Z 291.85,A -85,B 0,C 180,E1 -4208.247,E2 -4208.247} C_VEL
LIN {X 0,Y 530.993,Z 291.842,A -85,B 0,C 180,E1 -4210.678,E2 -4210.678} C_VEL
LIN {X 0,Y 530.987,Z 291.84,A -85,B 0,C 180,E1 -4213.071,E2 -4213.071} C_VEL
LIN {X 0,Y 531.015,Z 291.837,A -85,B 0,C 180,E1 -4215.436,E2 -4215.436} C_VEL
LIN {X 0,Y 531.034,Z 291.838,A -85,B 0,C 180,E1 -4218.55,E2 -4218.55} C_VEL
LIN {X 0,Y 531.052,Z 291.835,A -85,B 0,C 180,E1 -4221.63,E2 -4221.63} C_VEL
LIN {X 0,Y 531.119,Z 291.825,A -85,B 0,C 180,E1 -4224.685,E2 -4224.685} C_VEL
LIN {X 0,Y 531.139,Z 291.826,A -85,B 0,C 180,E1 -4227.725,E2 -4227.725} C_VEL
LIN {X 0,Y 531.15,Z 291.82,A -85,B 0,C 180,E1 -4230.758,E2 -4230.758} C_VEL
LIN {X 0,Y 531.102,Z 291.826,A -85,B 0,C 180,E1 -4233.034,E2 -4233.034} C_VEL
LIN {X 0,Y 531.083,Z 291.834,A -85,B 0,C 180,E1 -4236.077,E2 -4236.077} C_VEL
LIN {X 0,Y 531.027,Z 291.836,A -85,B 0,C 180,E1 -4239.138,E2 -4239.138} C_VEL
LIN {X 0,Y 531.037,Z 291.837,A -85,B 0,C 180,E1 -4242.225,E2 -4242.225} C_VEL
LIN {X 0,Y 530.992,Z 291.842,A -85,B 0,C 180,E1 -4245.349,E2 -4245.349} C_VEL
LIN {X 0,Y 531.013,Z 291.844,A -85,B 0,C 180,E1 -4247.722,E2 -4247.722} C_VEL
LIN {X 0,Y 530.995,Z 291.839,A -85,B 0,C 180,E1 -4250.938,E2 -4250.938} C_VEL
LIN {X 0,Y 530.975,Z 291.843,A -85,B 0,C 180,E1 -4254.224,E2 -4254.224} C_VEL
LIN {X 0,Y 531.007,Z 291.837,A -85,B 0,C 180,E1 -4256.743,E2 -4256.743} C_VEL
LIN {X 0,Y 530.977,Z 291.841,A -85,B 0,C 180,E1 -4259.322,E2 -4259.322} C_VEL
LIN {X 0,Y 530.975,Z 291.842,A -85,B 0,C 180,E1 -4262.103,E2 -4262.103} C_VEL
LIN {X 0,Y 530.984,Z 291.831,A -85,B 0,C 180,E1 -4264.854,E2 -4264.854} C_VEL
LIN {X 0,Y 530.959,Z 291.85,A -85,B 0,C 180,E1 -4267.507,E2 -4267.507} C_VEL
LIN {X 0,Y 530.977,Z 291.834,A -85,B 0,C 180,E1 -4270.432,E2 -4270.432} C_VEL
LIN {X 0,Y 530.962,Z 291.837,A -85,B 0,C 180,E1 -4273.282,E2 -4273.282} C_VEL
LIN {X 0,Y 530.98,Z 291.845,A -85,B 0,C 180,E1 -4275.62,E2 -4275.62} C_VEL
LIN {X 0,Y 530.998,Z 291.835,A -85,B 0,C 180,E1 -4278.566,E2 -4278.566} C_VEL
LIN {X 0,Y 530.959,Z 291.85,A -85,B 0,C 180,E1 -4281.346,E2 -4281.346} C_VEL
LIN {X 0,Y 530.973,Z 291.838,A -85,B 0,C 180,E1 -4284.382,E2 -4284.382} C_VEL
LIN {X 0,Y 530.965,Z 291.846,A -85,B 0,C 180,E1 -4287.134,E2 -4287.134} C_VEL
LIN {X 0,Y 530.976,Z 291.84,A -85,B 0,C 180,E1 -4289.804,E2 -4289.804} C_VEL
LIN {X 0,Y 531.006,Z 291.831,A -85,B 0,C 180,E1 -4292.467,E2 -4292.467} C_VEL
LIN {X 0,Y 530.995,Z 291.841,A -85,B 0,C 180,E1 -4294.942,E2 -4294.942} C_VEL
LIN {X 0,Y 530.961,Z 291.84,A -85,B 0,C 180,E1 -4298.247,E2 -4298.247} C_VEL
LIN {X 0,Y 530.987,Z 291.836,A -85,B 0,C 180,E1 -4300.677,E2 -4300.677} C_VEL
LIN {X 0,Y 530.983,Z 291.845,A -85,B 0,C 180,E1 -4303.071,E2 -4303.071} C_VEL
LIN {X 0,Y 531.008,Z 291.838,A -85,B 0,C 180,E1 -4305.436,E2 -4305.436} C_VEL
LIN {X 0,Y 531.036,Z 291.832,A -85,B 0,C 180,E1 -4308.55,E2 -4308.55} C_VEL
LIN {X 0,Y 531.047,Z 291.827,A -85,B 0,C 180,E1 -4311.63,E2 -4311.63} C_VEL
LIN {X 0,Y 531.113,Z 291.829,A -85,B 0,C 180,E1 -4314.686,E2 -4314.686} C_VEL
LIN {X 0,Y 531.128,Z 291.816,A -85,B 0,C 180,E1 -4317.725,E2 -4317.725} C_VEL
LIN {X 0,Y 531.147,Z 291.817,A -85,B 0,C 180,E1 -4320.759,E2 -4320.759} C_VEL
LIN {X 0,Y 531.099,Z 291.828,A -85,B 0,C 180,E1 -4323.035,E2 -4323.035} C_VEL
LIN {X 0,Y 531.073,Z 291.828,A -85,B 0,C 180,E1 -4326.078,E2 -4326.078} C_VEL
LIN {X 0,Y 531.026,Z 291.826,A -85,B 0,C 180,E1 -4329.139,E2 -4329.139} C_VEL
LIN {X 0,Y 531.032,Z 291.832,A -85,B 0,C 180,E1 -4332.226,E2 -4332.226} C_VEL
LIN {X 0,Y 530.987,Z 291.837,A -85,B 0,C 180,E1 -4335.35,E2 -4335.35} C_VEL
LIN {X 0,Y 530.983,Z 291.838,A -85,B 0,C 180,E1 -4338.522,E2 -4338.522} C_VEL
LIN {X 0,Y 530.994,Z 291.839,A -85,B 0,C 180,E1 -4340.939,E2 -4340.939} C_VEL
LIN {X 0,Y 530.958,Z 291.847,A -85,B 0,C 180,E1 -4344.226,E2 -4344.226} C_VEL
LIN {X 0,Y 530.998,Z 291.835,A -85,B 0,C 180,E1 -4346.744,E2 -4346.744} C_VEL
LIN {X 0,Y 530.975,Z 291.839,A -85,B 0,C 180,E1 -4349.323,E2 -4349.323} C_VEL
LIN {X 0,Y 530.958,Z 291.847,A -85,B 0,C 180,E1 -4352.101,E2 -4352.101} C_VEL
LIN {X 0,Y 530.963,Z 291.841,A -85,B 0,C 180,E1 -4354.852,E2 -4354.852} C_VEL
LIN {X 0,Y 530.96,Z 291.842,A -85,B 0,C 180,E1 -4357.509,E2 -4357.509} C_VEL
LIN {X 0,Y 530.976,Z 291.845,A -85,B 0,C 180,E1 -4360.434,E2 -4360.434} C_VEL
LIN {X 0,Y 530.956,Z 291.842,A -85,B 0,C 180,E1 -4363.282,E2 -4363.282} C_VEL
LIN {X 0,Y 530.973,Z 291.841,A -85,B 0,C 180,E1 -4365.623,E2 -4365.623} C_VEL
LIN {X 0,Y 530.99,Z 291.835,A -85,B 0,C 180,E1 -4368.565,E2 -4368.565} C_VEL
LIN {X 0,Y 530.952,Z 291.844,A -85,B 0,C 180,E1 -4371.53,E2 -4371.53} C_VEL
LIN {X 0,Y 530.948,Z 291.847,A -85,B 0,C 180,E1 -4374.38,E2 -4374.38} C_VEL
LIN {X 0,Y 530.966,Z 291.84,A -85,B 0,C 180,E1 -4377.134,E2 -4377.134} C_VEL
LIN {X 0,Y 530.968,Z 291.847,A -85,B 0,C 180,E1 -4379.804,E2 -4379.804} C_VEL
LIN {X 0,Y 531.008,Z 291.842,A -85,B 0,C 180,E1 -4382.469,E2 -4382.469} C_VEL
LIN {X 0,Y 531.018,Z 291.958,A -85,B 0,C 180,E1 -4384.156,E2 -4384.156} C_VEL
LIN {X 0,Y 532.123,Z 299.177,A -85,B 0,C 180,E1 -4385.689,E2 -4385.689} C_VEL
LIN {X 0,Y 531.738,Z 314.368,A -85,B 0,C 180,E1 -4388.687,E2 -4388.687} C_VEL
LIN {X 0,Y 531.44,Z 330.16,A -85,B 0,C 180,E1 -4391.715,E2 -4391.715} C_VEL
LIN {X 0,Y 531.149,Z 346.77,A -85,B 0,C 180,E1 -4394.876,E2 -4394.876} C_VEL
LIN {X 0,Y 531.123,Z 347.864,A -85,B 0,C 180,E1 -4395.038,E2 -4395.038} C_VEL
LIN {X 0,Y 532.834,Z 359.344,A -85,B 0,C 180,E1 -4395.27,E2 -4395.27} C_VEL
LIN {X 0,Y 532.424,Z 452.681,A -85,B 0,C 180,E1 -4396.547,E2 -4396.547} C_VEL
LIN {X 0,Y 532.268,Z 462.573,A -85,B 0,C 180,E1 -4396.762,E2 -4396.762} C_VEL
LIN {X 0,Y 532.14,Z 472.55,A -85,B 0,C 180,E1 -4397.074,E2 -4397.074} C_VEL
LIN {X 0,Y 531.973,Z 481.908,A -85,B 0,C 180,E1 -4397.458,E2 -4397.458} C_VEL
LIN {X 0,Y 531.753,Z 491.779,A -85,B 0,C 180,E1 -4397.969,E2 -4397.969} C_VEL
LIN {X 0,Y 531.558,Z 501.052,A -85,B 0,C 180,E1 -4398.561,E2 -4398.561} C_VEL
LIN {X 0,Y 531.363,Z 509.784,A -85,B 0,C 180,E1 -4399.233,E2 -4399.233} C_VEL
LIN {X 0,Y 531.161,Z 517.18,A -85,B 0,C 180,E1 -4399.903,E2 -4399.903} C_VEL
LIN {X 0,Y 531.003,Z 524.402,A -85,B 0,C 180,E1 -4400.67,E2 -4400.67} C_VEL
LIN {X 0,Y 530.87,Z 530.604,A -85,B 0,C 180,E1 -4401.435,E2 -4401.435} C_VEL
LIN {X 0,Y 530.703,Z 537.14,A -85,B 0,C 180,E1 -4402.39,E2 -4402.39} C_VEL
LIN {X 0,Y 530.57,Z 543.105,A -85,B 0,C 180,E1 -4403.446,E2 -4403.446} C_VEL
LIN {X 0,Y 530.587,Z 547.13,A -85,B 0,C 180,E1 -4404.299,E2 -4404.299} C_VEL
LIN {X 0,Y 530.459,Z 551.447,A -85,B 0,C 180,E1 -4405.441,E2 -4405.441} C_VEL
LIN {X 0,Y 530.516,Z 553.812,A -85,B 0,C 180,E1 -4406.202,E2 -4406.202} C_VEL
LIN {X 0,Y 530.457,Z 555.606,A -85,B 0,C 180,E1 -4406.962,E2 -4406.962} C_VEL
LIN {X 0,Y 530.361,Z 558.043,A -85,B 0,C 180,E1 -4408.481,E2 -4408.481} C_VEL
LIN {X 0,Y 530.344,Z 558.629,A -85,B 0,C 180,E1 -4409.241,E2 -4409.241} C_VEL
LIN {X 0,Y 530.344,Z 558.629,A -85,B 0,C 180,E1 -4410.759,E2 -4410.759} C_VEL
LIN {X 0,Y 530.361,Z 558.043,A -85,B 0,C 180,E1 -4411.519,E2 -4411.519} C_VEL
LIN {X 0,Y 530.457,Z 555.606,A -85,B 0,C 180,E1 -4413.038,E2 -4413.038} C_VEL
LIN {X 0,Y 530.524,Z 552.665,A -85,B 0,C 180,E1 -4414.178,E2 -4414.178} C_VEL
LIN {X 0,Y 530.523,Z 548.681,A -85,B 0,C 180,E1 -4415.321,E2 -4415.321} C_VEL
LIN {X 0,Y 530.542,Z 544.364,A -85,B 0,C 180,E1 -4416.304,E2 -4416.304} C_VEL
LIN {X 0,Y 530.666,Z 539.451,A -85,B 0,C 180,E1 -4417.228,E2 -4417.228} C_VEL
LIN {X 0,Y 530.784,Z 533.356,A -85,B 0,C 180,E1 -4418.183,E2 -4418.183} C_VEL
LIN {X 0,Y 530.912,Z 527.655,A -85,B 0,C 180,E1 -4418.948,E2 -4418.948} C_VEL
LIN {X 0,Y 531.106,Z 519.1,A -85,B 0,C 180,E1 -4419.905,E2 -4419.905} C_VEL
LIN {X 0,Y 531.341,Z 510.919,A -85,B 0,C 180,E1 -4420.671,E2 -4420.671} C_VEL
LIN {X 0,Y 531.53,Z 502.404,A -85,B 0,C 180,E1 -4421.343,E2 -4421.343} C_VEL
LIN {X 0,Y 531.718,Z 492.959,A -85,B 0,C 180,E1 -4421.961,E2 -4421.961} C_VEL
LIN {X 0,Y 531.937,Z 482.915,A -85,B 0,C 180,E1 -4422.494,E2 -4422.494} C_VEL
LIN {X 0,Y 532.133,Z 473.839,A -85,B 0,C 180,E1 -4422.877,E2 -4422.877} C_VEL
LIN {X 0,Y 532.248,Z 464.322,A -85,B 0,C 180,E1 -4423.19,E2 -4423.19} C_VEL
LIN {X 0,Y 532.418,Z 454.013,A -85,B 0,C 180,E1 -4423.429,E2 -4423.429} C_VEL
LIN {X 0,Y 532.649,Z 402.099,A -85,B 0,C 180,E1 -4424.152,E2 -4424.152} C_VEL
LIN {X 0,Y 532.72,Z 357.448,A -85,B 0,C 180,E1 -4424.759,E2 -4424.759} C_VEL
LIN {X 0,Y 531.141,Z 348.271,A -85,B 0,C 180,E1 -4424.939,E2 -4424.939} C_VEL
LIN {X 0,Y 531.116,Z 347.117,A -85,B 0,C 180,E1 -4425.057,E2 -4425.057} C_VEL
LIN {X 0,Y 531.409,Z 331.309,A -85,B 0,C 180,E1 -4428.067,E2 -4428.067} C_VEL
LIN {X 0,Y 531.738,Z 315.415,A -85,B 0,C 180,E1 -4431.11,E2 -4431.11} C_VEL
LIN {X 0,Y 532.088,Z 299.89,A -85,B 0,C 180,E1 -4434.17,E2 -4434.17} C_VEL
LIN {X 0,Y 531.71,Z 295.741,A -85,B 0,C 180,E1 -4435.021,E2 -4435.021} C_VEL
LIN {X 0,Y 531.021,Z 291.864,A -85,B 0,C 180,E1 -4435.896,E2 -4435.896} C_VEL
LIN {X 0,Y 530.971,Z 291.847,A -85,B 0,C 180,E1 -4438.456,E2 -4438.456} C_VEL
LIN {X 0,Y 530.956,Z 291.844,A -85,B 0,C 180,E1 -4441.078,E2 -4441.078} C_VEL
LIN {X 0,Y 530.986,Z 291.844,A -85,B 0,C 180,E1 -4443.772,E2 -4443.772} C_VEL
LIN {X 0,Y 530.948,Z 291.844,A -85,B 0,C 180,E1 -4446.558,E2 -4446.558} C_VEL
LIN {X 0,Y 530.982,Z 291.841,A -85,B 0,C 180,E1 -4449.443,E2 -4449.443} C_VEL
LIN {X 0,Y 530.974,Z 291.841,A -85,B 0,C 180,E1 -4452.456,E2 -4452.456} C_VEL
LIN {X 0,Y 530.973,Z 291.845,A -85,B 0,C 180,E1 -4455.621,E2 -4455.621} C_VEL
LIN {X 0,Y 530.995,Z 291.837,A -85,B 0,C 180,E1 -4458.564,E2 -4458.564} C_VEL
LIN {X 0,Y 530.952,Z 291.846,A -85,B 0,C 180,E1 -4461.528,E2 -4461.528} C_VEL
LIN {X 0,Y 530.948,Z 291.842,A -85,B 0,C 180,E1 -4464.379,E2 -4464.379} C_VEL
LIN {X 0,Y 530.96,Z 291.84,A -85,B 0,C 180,E1 -4467.132,E2 -4467.132} C_VEL
LIN {X 0,Y 530.962,Z 291.847,A -85,B 0,C 180,E1 -4469.802,E2 -4469.802} C_VEL
LIN {X 0,Y 531.009,Z 291.83,A -85,B 0,C 180,E1 -4472.466,E2 -4472.466} C_VEL
LIN {X 0,Y 530.987,Z 291.836,A -85,B 0,C 180,E1 -4474.941,E2 -4474.941} C_VEL
LIN {X 0,Y 530.963,Z 291.84,A -85,B 0,C 180,E1 -4478.246,E2 -4478.246} C_VEL
LIN {X 0,Y 530.987,Z 291.832,A -85,B 0,C 180,E1 -4480.677,E2 -4480.677} C_VEL
LIN {X 0,Y 530.978,Z 291.837,A -85,B 0,C 180,E1 -4483.07,E2 -4483.07} C_VEL
LIN {X 0,Y 531.031,Z 291.841,A -85,B 0,C 180,E1 -4485.436,E2 -4485.436} C_VEL
LIN {X 0,Y 531.037,Z 291.828,A -85,B 0,C 180,E1 -4488.549,E2 -4488.549} C_VEL
LIN {X 0,Y 531.05,Z 291.831,A -85,B 0,C 180,E1 -4491.629,E2 -4491.629} C_VEL
LIN {X 0,Y 531.114,Z 291.823,A -85,B 0,C 180,E1 -4494.685,E2 -4494.685} C_VEL
LIN {X 0,Y 531.127,Z 291.82,A -85,B 0,C 180,E1 -4497.725,E2 -4497.725} C_VEL
LIN {X 0,Y 531.146,Z 291.811,A -85,B 0,C 180,E1 -4500.758,E2 -4500.758} C_VEL
LIN {X 0,Y 531.1,Z 291.827,A -85,B 0,C 180,E1 -4503.034,E2 -4503.034} C_VEL
LIN {X 0,Y 531.073,Z 291.827,A -85,B 0,C 180,E1 -4506.077,E2 -4506.077} C_VEL
LIN {X 0,Y 531.023,Z 291.832,A -85,B 0,C 180,E1 -4509.138,E2 -4509.138} C_VEL
LIN {X 0,Y 531.03,Z 291.83,A -85,B 0,C 180,E1 -4512.225,E2 -4512.225} C_VEL
LIN {X 0,Y 530.985,Z 291.842,A -85,B 0,C 180,E1 -4515.35,E2 -4515.35} C_VEL
LIN {X 0,Y 530.98,Z 291.837,A -85,B 0,C 180,E1 -4518.521,E2 -4518.521} C_VEL
LIN {X 0,Y 530.992,Z 291.841,A -85,B 0,C 180,E1 -4520.938,E2 -4520.938} C_VEL
LIN {X 0,Y 530.969,Z 291.841,A -85,B 0,C 180,E1 -4524.224,E2 -4524.224} C_VEL
LIN {X 0,Y 530.995,Z 291.84,A -85,B 0,C 180,E1 -4526.744,E2 -4526.744} C_VEL
LIN {X 0,Y 530.99,Z 291.839,A -85,B 0,C 180,E1 -4529.322,E2 -4529.322} C_VEL
LIN {X 0,Y 530.97,Z 291.841,A -85,B 0,C 180,E1 -4532.103,E2 -4532.103} C_VEL
LIN {X 0,Y 530.982,Z 291.842,A -85,B 0,C 180,E1 -4534.855,E2 -4534.855} C_VEL
LIN {X 0,Y 530.957,Z 291.843,A -85,B 0,C 180,E1 -4537.508,E2 -4537.508} C_VEL
LIN {X 0,Y 531.017,Z 291.838,A -85,B 0,C 180,E1 -4540.429,E2 -4540.429} C_VEL
LIN {X 0,Y 530.953,Z 291.842,A -85,B 0,C 180,E1 -4543.578,E2 -4543.578} C_VEL
LIN {X 0,Y 530.282,Z 291.931,A -85,B 0,C 180,E1 -4544.211,E2 -4544.211} C_VEL
LIN {X 0,Y 527.435,Z 292.282,A -85,B 0,C 180,E1 -4545.24,E2 -4545.24} C_VEL
LIN {X 0,Y 525.032,Z 292.579,A -85,B 0,C 180,E1 -4546.069,E2 -4546.069} C_VEL
LIN {X 0,Y 523.999,Z 292.704,A -85,B 0,C 180,E1 -4546.708,E2 -4546.708} C_VEL
LIN {X 0,Y 523.914,Z 292.71,A -85,B 0,C 180,E1 -4546.925,E2 -4546.925} C_VEL
LIN {X 0,Y 523.94,Z 292.712,A -85,B 0,C 180,E1 -4549.921,E2 -4549.921} C_VEL
LIN {X 0,Y 523.904,Z 292.723,A -85,B 0,C 180,E1 -4552.869,E2 -4552.869} C_VEL
LIN {X 0,Y 523.939,Z 292.708,A -85,B 0,C 180,E1 -4555.711,E2 -4555.711} C_VEL
LIN {X 0,Y 523.926,Z 292.726,A -85,B 0,C 180,E1 -4558.457,E2 -4558.457} C_VEL
LIN {X 0,Y 523.934,Z 292.715,A -85,B 0,C 180,E1 -4561.126,E2 -4561.126} C_VEL
LIN {X 0,Y 523.981,Z 292.716,A -85,B 0,C 180,E1 -4563.98,E2 -4563.98} C_VEL
LIN {X 0,Y 523.932,Z 292.726,A -85,B 0,C 180,E1 -4566.271,E2 -4566.271} C_VEL
LIN {X 0,Y 523.941,Z 292.72,A -85,B 0,C 180,E1 -4568.767,E2 -4568.767} C_VEL
LIN {X 0,Y 523.949,Z 292.716,A -85,B 0,C 180,E1 -4571.221,E2 -4571.221} C_VEL
LIN {X 0,Y 523.935,Z 292.72,A -85,B 0,C 180,E1 -4573.639,E2 -4573.639} C_VEL
LIN {X 0,Y 523.937,Z 292.724,A -85,B 0,C 180,E1 -4576.028,E2 -4576.028} C_VEL
LIN {X 0,Y 524.008,Z 292.715,A -85,B 0,C 180,E1 -4578.394,E2 -4578.394} C_VEL
LIN {X 0,Y 524,Z 292.712,A -85,B 0,C 180,E1 -4581.516,E2 -4581.516} C_VEL
LIN {X 0,Y 524.08,Z 292.703,A -85,B 0,C 180,E1 -4584.614,E2 -4584.614} C_VEL
LIN {X 0,Y 524.111,Z 292.701,A -85,B 0,C 180,E1 -4587.695,E2 -4587.695} C_VEL
LIN {X 0,Y 524.12,Z 292.696,A -85,B 0,C 180,E1 -4590.768,E2 -4590.768} C_VEL
LIN {X 0,Y 524.069,Z 292.702,A -85,B 0,C 180,E1 -4593.075,E2 -4593.075} C_VEL
LIN {X 0,Y 524.045,Z 292.71,A -85,B 0,C 180,E1 -4596.159,E2 -4596.159} C_VEL
LIN {X 0,Y 523.995,Z 292.713,A -85,B 0,C 180,E1 -4599.262,E2 -4599.262} C_VEL
LIN {X 0,Y 523.999,Z 292.717,A -85,B 0,C 180,E1 -4601.74,E2 -4601.74} C_VEL
LIN {X 0,Y 523.989,Z 292.713,A -85,B 0,C 180,E1 -4605.052,E2 -4605.052} C_VEL
LIN {X 0,Y 523.96,Z 292.721,A -85,B 0,C 180,E1 -4607.969,E2 -4607.969} C_VEL
LIN {X 0,Y 523.967,Z 292.715,A -85,B 0,C 180,E1 -4610.41,E2 -4610.41} C_VEL
LIN {X 0,Y 523.912,Z 292.721,A -85,B 0,C 180,E1 -4612.893,E2 -4612.893} C_VEL
LIN {X 0,Y 523.95,Z 292.722,A -85,B 0,C 180,E1 -4615.418,E2 -4615.418} C_VEL
LIN {X 0,Y 523.965,Z 292.714,A -85,B 0,C 180,E1 -4617.998,E2 -4617.998} C_VEL
LIN {X 0,Y 523.941,Z 292.716,A -85,B 0,C 180,E1 -4620.855,E2 -4620.855} C_VEL
LIN {X 0,Y 523.956,Z 292.711,A -85,B 0,C 180,E1 -4623.735,E2 -4623.735} C_VEL
LIN {X 0,Y 523.915,Z 292.718,A -85,B 0,C 180,E1 -4626.404,E2 -4626.404} C_VEL
LIN {X 0,Y 523.916,Z 292.723,A -85,B 0,C 180,E1 -4629.084,E2 -4629.084} C_VEL
LIN {X 0,Y 523.949,Z 292.703,A -85,B 0,C 180,E1 -4632.118,E2 -4632.118} C_VEL
LIN {X 0,Y 523.948,Z 292.72,A -85,B 0,C 180,E1 -4635.308,E2 -4635.308} C_VEL
LIN {X 0,Y 523.963,Z 292.712,A -85,B 0,C 180,E1 -4638.687,E2 -4638.687} C_VEL
LIN {X 0,Y 523.916,Z 292.723,A -85,B 0,C 180,E1 -4641.079,E2 -4641.079} C_VEL
LIN {X 0,Y 523.918,Z 292.718,A -85,B 0,C 180,E1 -4643.827,E2 -4643.827} C_VEL
LIN {X 0,Y 523.934,Z 292.715,A -85,B 0,C 180,E1 -4646.636,E2 -4646.636} C_VEL
LIN {X 0,Y 523.954,Z 292.72,A -85,B 0,C 180,E1 -4649.356,E2 -4649.356} C_VEL
LIN {X 0,Y 523.969,Z 292.706,A -85,B 0,C 180,E1 -4652.281,E2 -4652.281} C_VEL
LIN {X 0,Y 523.942,Z 292.715,A -85,B 0,C 180,E1 -4654.581,E2 -4654.581} C_VEL
LIN {X 0,Y 523.906,Z 292.728,A -85,B 0,C 180,E1 -4657.107,E2 -4657.107} C_VEL
LIN {X 0,Y 523.968,Z 292.706,A -85,B 0,C 180,E1 -4659.866,E2 -4659.866} C_VEL
LIN {X 0,Y 523.961,Z 292.715,A -85,B 0,C 180,E1 -4662.838,E2 -4662.838} C_VEL
LIN {X 0,Y 523.966,Z 292.718,A -85,B 0,C 180,E1 -4665.236,E2 -4665.236} C_VEL
LIN {X 0,Y 524.001,Z 292.707,A -85,B 0,C 180,E1 -4668.394,E2 -4668.394} C_VEL
LIN {X 0,Y 523.995,Z 292.706,A -85,B 0,C 180,E1 -4671.516,E2 -4671.516} C_VEL
LIN {X 0,Y 524.074,Z 292.704,A -85,B 0,C 180,E1 -4674.614,E2 -4674.614} C_VEL
LIN {X 0,Y 524.1,Z 292.692,A -85,B 0,C 180,E1 -4677.695,E2 -4677.695} C_VEL
LIN {X 0,Y 524.117,Z 292.692,A -85,B 0,C 180,E1 -4680.769,E2 -4680.769} C_VEL
LIN {X 0,Y 524.065,Z 292.704,A -85,B 0,C 180,E1 -4683.075,E2 -4683.075} C_VEL
LIN {X 0,Y 524.036,Z 292.705,A -85,B 0,C 180,E1 -4686.16,E2 -4686.16} C_VEL
LIN {X 0,Y 523.994,Z 292.7,A -85,B 0,C 180,E1 -4689.262,E2 -4689.262} C_VEL
LIN {X 0,Y 523.999,Z 292.705,A -85,B 0,C 180,E1 -4691.743,E2 -4691.743} C_VEL
LIN {X 0,Y 523.985,Z 292.711,A -85,B 0,C 180,E1 -4695.053,E2 -4695.053} C_VEL
LIN {X 0,Y 523.955,Z 292.709,A -85,B 0,C 180,E1 -4697.97,E2 -4697.97} C_VEL
LIN {X 0,Y 523.964,Z 292.714,A -85,B 0,C 180,E1 -4700.411,E2 -4700.411} C_VEL
LIN {X 0,Y 523.903,Z 292.723,A -85,B 0,C 180,E1 -4702.894,E2 -4702.894} C_VEL
LIN {X 0,Y 523.977,Z 292.711,A -85,B 0,C 180,E1 -4706.021,E2 -4706.021} C_VEL
LIN {X 0,Y 523.933,Z 292.718,A -85,B 0,C 180,E1 -4708.875,E2 -4708.875} C_VEL
LIN {X 0,Y 523.913,Z 292.719,A -85,B 0,C 180,E1 -4711.545,E2 -4711.545} C_VEL
LIN {X 0,Y 523.915,Z 292.721,A -85,B 0,C 180,E1 -4714.292,E2 -4714.292} C_VEL
LIN {X 0,Y 523.901,Z 292.721,A -85,B 0,C 180,E1 -4717.133,E2 -4717.133} C_VEL
LIN {X 0,Y 523.933,Z 292.721,A -85,B 0,C 180,E1 -4720.131,E2 -4720.131} C_VEL
LIN {X 0,Y 523.932,Z 292.722,A -85,B 0,C 180,E1 -4722.46,E2 -4722.46} C_VEL
LIN {X 0,Y 523.94,Z 292.716,A -85,B 0,C 180,E1 -4725.311,E2 -4725.311} C_VEL
LIN {X 0,Y 523.952,Z 292.71,A -85,B 0,C 180,E1 -4728.691,E2 -4728.691} C_VEL
LIN {X 0,Y 523.913,Z 292.719,A -85,B 0,C 180,E1 -4731.082,E2 -4731.082} C_VEL
LIN {X 0,Y 523.893,Z 292.726,A -85,B 0,C 180,E1 -4733.826,E2 -4733.826} C_VEL
LIN {X 0,Y 523.94,Z 292.717,A -85,B 0,C 180,E1 -4736.636,E2 -4736.636} C_VEL
LIN {X 0,Y 523.955,Z 292.718,A -85,B 0,C 180,E1 -4739.356,E2 -4739.356} C_VEL
LIN {X 0,Y 523.972,Z 292.718,A -85,B 0,C 180,E1 -4742.283,E2 -4742.283} C_VEL
LIN {X 0,Y 523.989,Z 292.821,A -85,B 0,C 180,E1 -4743.98,E2 -4743.98} C_VEL
LIN {X 0,Y 525.117,Z 299.902,A -85,B 0,C 180,E1 -4745.519,E2 -4745.519} C_VEL
LIN {X 0,Y 524.794,Z 314.232,A -85,B 0,C 180,E1 -4748.391,E2 -4748.391} C_VEL
LIN {X 0,Y 524.427,Z 330.967,A -85,B 0,C 180,E1 -4751.644,E2 -4751.644} C_VEL
LIN {X 0,Y 524.108,Z 347.585,A -85,B 0,C 180,E1 -4754.827,E2 -4754.827} C_VEL
LIN {X 0,Y 525.224,Z 354.722,A -85,B 0,C 180,E1 -4754.991,E2 -4754.991} C_VEL
LIN {X 0,Y 525.947,Z 360.285,A -85,B 0,C 180,E1 -4755.088,E2 -4755.088} C_VEL
LIN {X 0,Y 525.545,Z 452.488,A -85,B 0,C 180,E1 -4756.368,E2 -4756.368} C_VEL
LIN {X 0,Y 525.373,Z 462.379,A -85,B 0,C 180,E1 -4756.585,E2 -4756.585} C_VEL
LIN {X 0,Y 525.22,Z 472.356,A -85,B 0,C 180,E1 -4756.901,E2 -4756.901} C_VEL
LIN {X 0,Y 525.011,Z 481.713,A -85,B 0,C 180,E1 -4757.289,E2 -4757.289} C_VEL
LIN {X 0,Y 524.776,Z 491.676,A -85,B 0,C 180,E1 -4757.813,E2 -4757.813} C_VEL
LIN {X 0,Y 524.584,Z 500.858,A -85,B 0,C 180,E1 -4758.407,E2 -4758.407} C_VEL
LIN {X 0,Y 524.361,Z 509.589,A -85,B 0,C 180,E1 -4759.087,E2 -4759.087} C_VEL
LIN {X 0,Y 524.146,Z 516.986,A -85,B 0,C 180,E1 -4759.767,E2 -4759.767} C_VEL
LIN {X 0,Y 523.971,Z 524.207,A -85,B 0,C 180,E1 -4760.543,E2 -4760.543} C_VEL
LIN {X 0,Y 523.803,Z 530.409,A -85,B 0,C 180,E1 -4761.319,E2 -4761.319} C_VEL
LIN {X 0,Y 523.648,Z 536.946,A -85,B 0,C 180,E1 -4762.287,E2 -4762.287} C_VEL
LIN {X 0,Y 523.565,Z 541.447,A -85,B 0,C 180,E1 -4763.061,E2 -4763.061} C_VEL
LIN {X 0,Y 523.499,Z 546.935,A -85,B 0,C 180,E1 -4764.221,E2 -4764.221} C_VEL
LIN {X 0,Y 523.364,Z 551.253,A -85,B 0,C 180,E1 -4765.379,E2 -4765.379} C_VEL
LIN {X 0,Y 523.444,Z 553.619,A -85,B 0,C 180,E1 -4766.151,E2 -4766.151} C_VEL
LIN {X 0,Y 523.368,Z 555.412,A -85,B 0,C 180,E1 -4766.921,E2 -4766.921} C_VEL
LIN {X 0,Y 523.275,Z 557.849,A -85,B 0,C 180,E1 -4768.461,E2 -4768.461} C_VEL
LIN {X 0,Y 523.25,Z 558.436,A -85,B 0,C 180,E1 -4769.23,E2 -4769.23} C_VEL
LIN {X 0,Y 523.25,Z 558.436,A -85,B 0,C 180,E1 -4770.77,E2 -4770.77} C_VEL
LIN {X 0,Y 523.275,Z 557.849,A -85,B 0,C 180,E1 -4771.539,E2 -4771.539} C_VEL
LIN {X 0,Y 523.368,Z 555.412,A -85,B 0,C 180,E1 -4773.079,E2 -4773.079} C_VEL
LIN {X 0,Y 523.426,Z 552.47,A -85,B 0,C 180,E1 -4774.235,E2 -4774.235} C_VEL
LIN {X 0,Y 523.459,Z 548.487,A -85,B 0,C 180,E1 -4775.393,E2 -4775.393} C_VEL
LIN {X 0,Y 523.512,Z 543.276,A -85,B 0,C 180,E1 -4776.569,E2 -4776.569} C_VEL
LIN {X 0,Y 523.606,Z 538.101,A -85,B 0,C 180,E1 -4777.52,E2 -4777.52} C_VEL
LIN {X 0,Y 523.765,Z 531.785,A -85,B 0,C 180,E1 -4778.488,E2 -4778.488} C_VEL
LIN {X 0,Y 523.919,Z 525.834,A -85,B 0,C 180,E1 -4779.263,E2 -4779.263} C_VEL
LIN {X 0,Y 524.068,Z 518.905,A -85,B 0,C 180,E1 -4780.04,E2 -4780.04} C_VEL
LIN {X 0,Y 524.338,Z 510.724,A -85,B 0,C 180,E1 -4780.815,E2 -4780.815} C_VEL
LIN {X 0,Y 524.547,Z 502.21,A -85,B 0,C 180,E1 -4781.496,E2 -4781.496} C_VEL
LIN {X 0,Y 524.725,Z 493.827,A -85,B 0,C 180,E1 -4782.059,E2 -4782.059} C_VEL
LIN {X 0,Y 524.974,Z 483.728,A -85,B 0,C 180,E1 -4782.614,E2 -4782.614} C_VEL
LIN {X 0,Y 525.183,Z 474.933,A -85,B 0,C 180,E1 -4783.002,E2 -4783.002} C_VEL
LIN {X 0,Y 525.321,Z 465.003,A -85,B 0,C 180,E1 -4783.343,E2 -4783.343} C_VEL
LIN {X 0,Y 525.492,Z 455.151,A -85,B 0,C 180,E1 -4783.584,E2 -4783.584} C_VEL
LIN {X 0,Y 525.677,Z 432.336,A -85,B 0,C 180,E1 -4783.925,E2 -4783.925} C_VEL
LIN {X 0,Y 525.784,Z 357.913,A -85,B 0,C 180,E1 -4784.949,E2 -4784.949} C_VEL
LIN {X 0,Y 524.106,Z 347.825,A -85,B 0,C 180,E1 -4785.156,E2 -4785.156} C_VEL
LIN {X 0,Y 524.078,Z 346.814,A -85,B 0,C 180,E1 -4785.285,E2 -4785.285} C_VEL
LIN {X 0,Y 524.427,Z 330.967,A -85,B 0,C 180,E1 -4788.356,E2 -4788.356} C_VEL
LIN {X 0,Y 524.748,Z 315.279,A -85,B 0,C 180,E1 -4791.405,E2 -4791.405} C_VEL
LIN {X 0,Y 525.147,Z 300.428,A -85,B 0,C 180,E1 -4794.373,E2 -4794.373} C_VEL
LIN {X 0,Y 523.969,Z 292.773,A -85,B 0,C 180,E1 -4796.042,E2 -4796.042} C_VEL
LIN {X 0,Y 523.928,Z 292.721,A -85,B 0,C 180,E1 -4798.875,E2 -4798.875} C_VEL
LIN {X 0,Y 523.92,Z 292.724,A -85,B 0,C 180,E1 -4801.543,E2 -4801.543} C_VEL
LIN {X 0,Y 523.93,Z 292.721,A -85,B 0,C 180,E1 -4804.289,E2 -4804.289} C_VEL
LIN {X 0,Y 523.902,Z 292.721,A -85,B 0,C 180,E1 -4807.132,E2 -4807.132} C_VEL
LIN {X 0,Y 523.935,Z 292.715,A -85,B 0,C 180,E1 -4810.129,E2 -4810.129} C_VEL
LIN {X 0,Y 523.931,Z 292.719,A -85,B 0,C 180,E1 -4812.458,E2 -4812.458} C_VEL
LIN {X 0,Y 523.94,Z 292.718,A -85,B 0,C 180,E1 -4815.309,E2 -4815.309} C_VEL
LIN {X 0,Y 523.957,Z 292.713,A -85,B 0,C 180,E1 -4818.688,E2 -4818.688} C_VEL
LIN {X 0,Y 523.91,Z 292.727,A -85,B 0,C 180,E1 -4821.897,E2 -4821.897} C_VEL
LIN {X 0,Y 523.918,Z 292.717,A -85,B 0,C 180,E1 -4824.91,E2 -4824.91} C_VEL
LIN {X 0,Y 523.928,Z 292.723,A -85,B 0,C 180,E1 -4827.679,E2 -4827.679} C_VEL
LIN {X 0,Y 523.947,Z 292.714,A -85,B 0,C 180,E1 -4830.676,E2 -4830.676} C_VEL
LIN {X 0,Y 523.967,Z 292.714,A -85,B 0,C 180,E1 -4833.728,E2 -4833.728} C_VEL
LIN {X 0,Y 523.917,Z 292.719,A -85,B 0,C 180,E1 -4836.269,E2 -4836.269} C_VEL
LIN {X 0,Y 523.939,Z 292.715,A -85,B 0,C 180,E1 -4838.766,E2 -4838.766} C_VEL
LIN {X 0,Y 523.944,Z 292.714,A -85,B 0,C 180,E1 -4841.22,E2 -4841.22} C_VEL
LIN {X 0,Y 523.93,Z 292.722,A -85,B 0,C 180,E1 -4843.638,E2 -4843.638} C_VEL
LIN {X 0,Y 523.937,Z 292.717,A -85,B 0,C 180,E1 -4846.028,E2 -4846.028} C_VEL
LIN {X 0,Y 524.003,Z 292.704,A -85,B 0,C 180,E1 -4848.393,E2 -4848.393} C_VEL
LIN {X 0,Y 523.998,Z 292.71,A -85,B 0,C 180,E1 -4851.515,E2 -4851.515} C_VEL
LIN {X 0,Y 524.075,Z 292.699,A -85,B 0,C 180,E1 -4854.613,E2 -4854.613} C_VEL
LIN {X 0,Y 524.099,Z 292.695,A -85,B 0,C 180,E1 -4857.694,E2 -4857.694} C_VEL
LIN {X 0,Y 524.116,Z 292.686,A -85,B 0,C 180,E1 -4860.768,E2 -4860.768} C_VEL
LIN {X 0,Y 524.066,Z 292.703,A -85,B 0,C 180,E1 -4863.075,E2 -4863.075} C_VEL
LIN {X 0,Y 524.035,Z 292.704,A -85,B 0,C 180,E1 -4866.159,E2 -4866.159} C_VEL
LIN {X 0,Y 523.991,Z 292.705,A -85,B 0,C 180,E1 -4869.262,E2 -4869.262} C_VEL
LIN {X 0,Y 523.998,Z 292.706,A -85,B 0,C 180,E1 -4871.742,E2 -4871.742} C_VEL
LIN {X 0,Y 523.981,Z 292.719,A -85,B 0,C 180,E1 -4875.052,E2 -4875.052} C_VEL
LIN {X 0,Y 523.953,Z 292.709,A -85,B 0,C 180,E1 -4877.969,E2 -4877.969} C_VEL
LIN {X 0,Y 523.962,Z 292.709,A -85,B 0,C 180,E1 -4880.41,E2 -4880.41} C_VEL
LIN {X 0,Y 523.906,Z 292.728,A -85,B 0,C 180,E1 -4882.893,E2 -4882.893} C_VEL
LIN {X 0,Y 523.942,Z 292.715,A -85,B 0,C 180,E1 -4885.419,E2 -4885.419} C_VEL
LIN {X 0,Y 523.96,Z 292.708,A -85,B 0,C 180,E1 -4887.999,E2 -4887.999} C_VEL
LIN {X 0,Y 523.943,Z 292.724,A -85,B 0,C 180,E1 -4890.856,E2 -4890.856} C_VEL
LIN {X 0,Y 523.953,Z 292.711,A -85,B 0,C 180,E1 -4893.735,E2 -4893.735} C_VEL
LIN {X 0,Y 523.913,Z 292.721,A -85,B 0,C 180,E1 -4896.405,E2 -4896.405} C_VEL
LIN {X 0,Y 523.923,Z 292.72,A -85,B 0,C 180,E1 -4899.084,E2 -4899.084} C_VEL
LIN {X 0,Y 523.963,Z 292.712,A -85,B 0,C 180,E1 -4901.313,E2 -4901.313} C_VEL
LIN {X 0,Y 523.948,Z 292.72,A -85,B 0,C 180,E1 -4904.692,E2 -4904.692} C_VEL
LIN {X 0,Y 523.914,Z 292.71,A -85,B 0,C 180,E1 -4906.925,E2 -4906.925} C_VEL
LIN {X 0,Y 523.247,Z 292.79,A -85,B 0,C 180,E1 -4907.566,E2 -4907.566} C_VEL
LIN {X 0,Y 520.402,Z 293.15,A -85,B 0,C 180,E1 -4908.608,E2 -4908.608} C_VEL
LIN {X 0,Y 517.996,Z 293.453,A -85,B 0,C 180,E1 -4909.447,E2 -4909.447} C_VEL
LIN {X 0,Y 516.96,Z 293.584,A -85,B 0,C 180,E1 -4910.095,E2 -4910.095} C_VEL
LIN {X 0,Y 516.874,Z 293.596,A -85,B 0,C 180,E1 -4910.314,E2 -4910.314} C_VEL
LIN {X 0,Y 516.878,Z 293.595,A -85,B 0,C 180,E1 -4913.342,E2 -4913.342} C_VEL
LIN {X 0,Y 516.907,Z 293.587,A -85,B 0,C 180,E1 -4916.122,E2 -4916.122} C_VEL
LIN {X 0,Y 516.886,Z 293.596,A -85,B 0,C 180,E1 -4918.936,E2 -4918.936} C_VEL
LIN {X 0,Y 516.914,Z 293.589,A -85,B 0,C 180,E1 -4921.585,E2 -4921.585} C_VEL
LIN {X 0,Y 516.928,Z 293.598,A -85,B 0,C 180,E1 -4924.211,E2 -4924.211} C_VEL
LIN {X 0,Y 516.867,Z 293.601,A -85,B 0,C 180,E1 -4926.777,E2 -4926.777} C_VEL
LIN {X 0,Y 516.934,Z 293.592,A -85,B 0,C 180,E1 -4929.732,E2 -4929.732} C_VEL
LIN {X 0,Y 516.927,Z 293.595,A -85,B 0,C 180,E1 -4932.597,E2 -4932.597} C_VEL
LIN {X 0,Y 516.938,Z 293.591,A -85,B 0,C 180,E1 -4935.03,E2 -4935.03} C_VEL
LIN {X 0,Y 516.962,Z 293.594,A -85,B 0,C 180,E1 -4938.234,E2 -4938.234} C_VEL
LIN {X 0,Y 516.965,Z 293.588,A -85,B 0,C 180,E1 -4941.4,E2 -4941.4} C_VEL
LIN {X 0,Y 517.009,Z 293.586,A -85,B 0,C 180,E1 -4943.757,E2 -4943.757} C_VEL
LIN {X 0,Y 517.082,Z 293.576,A -85,B 0,C 180,E1 -4947.663,E2 -4947.663} C_VEL
LIN {X 0,Y 517.091,Z 293.572,A -85,B 0,C 180,E1 -4950.779,E2 -4950.779} C_VEL
LIN {X 0,Y 517.01,Z 293.582,A -85,B 0,C 180,E1 -4953.117,E2 -4953.117} C_VEL
LIN {X 0,Y 517.009,Z 293.586,A -85,B 0,C 180,E1 -4956.243,E2 -4956.243} C_VEL
LIN {X 0,Y 516.95,Z 293.592,A -85,B 0,C 180,E1 -4959.389,E2 -4959.389} C_VEL
LIN {X 0,Y 516.949,Z 293.596,A -85,B 0,C 180,E1 -4961.807,E2 -4961.807} C_VEL
LIN {X 0,Y 516.94,Z 293.591,A -85,B 0,C 180,E1 -4965.146,E2 -4965.146} C_VEL
LIN {X 0,Y 516.922,Z 293.595,A -85,B 0,C 180,E1 -4968.222,E2 -4968.222} C_VEL
LIN {X 0,Y 516.908,Z 293.594,A -85,B 0,C 180,E1 -4970.701,E2 -4970.701} C_VEL
LIN {X 0,Y 516.906,Z 293.597,A -85,B 0,C 180,E1 -4974.072,E2 -4974.072} C_VEL
LIN {X 0,Y 516.924,Z 293.591,A -85,B 0,C 180,E1 -4976.657,E2 -4976.657} C_VEL
LIN {X 0,Y 516.905,Z 293.593,A -85,B 0,C 180,E1 -4979.524,E2 -4979.524} C_VEL
LIN {X 0,Y 516.895,Z 293.594,A -85,B 0,C 180,E1 -4982.544,E2 -4982.544} C_VEL
LIN {X 0,Y 516.876,Z 293.592,A -85,B 0,C 180,E1 -4985.332,E2 -4985.332} C_VEL
LIN {X 0,Y 516.874,Z 293.6,A -85,B 0,C 180,E1 -4987.943,E2 -4987.943} C_VEL
LIN {X 0,Y 516.878,Z 293.591,A -85,B 0,C 180,E1 -4990.741,E2 -4990.741} C_VEL
LIN {X 0,Y 516.896,Z 293.581,A -85,B 0,C 180,E1 -4992.829,E2 -4992.829} C_VEL
LIN {X 0,Y 516.914,Z 293.591,A -85,B 0,C 180,E1 -4995.01,E2 -4995.01} C_VEL
LIN {X 0,Y 516.914,Z 293.589,A -85,B 0,C 180,E1 -4998.397,E2 -4998.397} C_VEL
LIN {X 0,Y 516.877,Z 293.603,A -85,B 0,C 180,E1 -5001.284,E2 -5001.284} C_VEL
LIN {X 0,Y 516.881,Z 293.593,A -85,B 0,C 180,E1 -5004.221,E2 -5004.221} C_VEL
LIN {X 0,Y 516.889,Z 293.597,A -85,B 0,C 180,E1 -5007.053,E2 -5007.053} C_VEL
LIN {X 0,Y 516.892,Z 293.595,A -85,B 0,C 180,E1 -5009.797,E2 -5009.797} C_VEL
LIN {X 0,Y 516.918,Z 293.585,A -85,B 0,C 180,E1 -5012.467,E2 -5012.467} C_VEL
LIN {X 0,Y 516.9,Z 293.598,A -85,B 0,C 180,E1 -5015.072,E2 -5015.072} C_VEL
LIN {X 0,Y 516.876,Z 293.596,A -85,B 0,C 180,E1 -5018.462,E2 -5018.462} C_VEL
LIN {X 0,Y 516.894,Z 293.592,A -85,B 0,C 180,E1 -5020.955,E2 -5020.955} C_VEL
LIN {X 0,Y 516.907,Z 293.594,A -85,B 0,C 180,E1 -5023.41,E2 -5023.41} C_VEL
LIN {X 0,Y 516.885,Z 293.595,A -85,B 0,C 180,E1 -5025.834,E2 -5025.834} C_VEL
LIN {X 0,Y 516.954,Z 293.583,A -85,B 0,C 180,E1 -5028.234,E2 -5028.234} C_VEL
LIN {X 0,Y 516.96,Z 293.583,A -85,B 0,C 180,E1 -5031.4,E2 -5031.4} C_VEL
LIN {X 0,Y 516.999,Z 293.58,A -85,B 0,C 180,E1 -5033.757,E2 -5033.757} C_VEL
LIN {X 0,Y 517.073,Z 293.567,A -85,B 0,C 180,E1 -5037.664,E2 -5037.664} C_VEL
LIN {X 0,Y 517.087,Z 293.567,A -85,B 0,C 180,E1 -5040.779,E2 -5040.779} C_VEL
LIN {X 0,Y 517.006,Z 293.583,A -85,B 0,C 180,E1 -5043.117,E2 -5043.117} C_VEL
LIN {X 0,Y 517,Z 293.583,A -85,B 0,C 180,E1 -5046.244,E2 -5046.244} C_VEL
LIN {X 0,Y 516.948,Z 293.576,A -85,B 0,C 180,E1 -5049.39,E2 -5049.39} C_VEL
LIN {X 0,Y 516.948,Z 293.583,A -85,B 0,C 180,E1 -5051.811,E2 -5051.811} C_VEL
LIN {X 0,Y 516.938,Z 293.588,A -85,B 0,C 180,E1 -5055.148,E2 -5055.148} C_VEL
LIN {X 0,Y 516.917,Z 293.588,A -85,B 0,C 180,E1 -5058.223,E2 -5058.223} C_VEL
LIN {X 0,Y 516.905,Z 293.597,A -85,B 0,C 180,E1 -5060.702,E2 -5060.702} C_VEL
LIN {X 0,Y 516.879,Z 293.599,A -85,B 0,C 180,E1 -5064.074,E2 -5064.074} C_VEL
LIN {X 0,Y 516.919,Z 293.589,A -85,B 0,C 180,E1 -5066.659,E2 -5066.659} C_VEL
LIN {X 0,Y 516.904,Z 293.592,A -85,B 0,C 180,E1 -5069.525,E2 -5069.525} C_VEL
LIN {X 0,Y 516.887,Z 293.596,A -85,B 0,C 180,E1 -5072.544,E2 -5072.544} C_VEL
LIN {X 0,Y 516.86,Z 293.595,A -85,B 0,C 180,E1 -5075.331,E2 -5075.331} C_VEL
LIN {X 0,Y 516.875,Z 293.601,A -85,B 0,C 180,E1 -5077.944,E2 -5077.944} C_VEL
LIN {X 0,Y 516.879,Z 293.597,A -85,B 0,C 180,E1 -5080.743,E2 -5080.743} C_VEL
LIN {X 0,Y 516.878,Z 293.597,A -85,B 0,C 180,E1 -5082.832,E2 -5082.832} C_VEL
LIN {X 0,Y 516.891,Z 293.594,A -85,B 0,C 180,E1 -5085.008,E2 -5085.008} C_VEL
LIN {X 0,Y 516.91,Z 293.59,A -85,B 0,C 180,E1 -5088.4,E2 -5088.4} C_VEL
LIN {X 0,Y 516.877,Z 293.596,A -85,B 0,C 180,E1 -5091.285,E2 -5091.285} C_VEL
LIN {X 0,Y 516.866,Z 293.6,A -85,B 0,C 180,E1 -5094.22,E2 -5094.22} C_VEL
LIN {X 0,Y 516.894,Z 293.593,A -85,B 0,C 180,E1 -5097.054,E2 -5097.054} C_VEL
LIN {X 0,Y 516.891,Z 293.6,A -85,B 0,C 180,E1 -5099.797,E2 -5099.797} C_VEL
LIN {X 0,Y 516.922,Z 293.598,A -85,B 0,C 180,E1 -5102.468,E2 -5102.468} C_VEL
LIN {X 0,Y 516.967,Z 293.823,A -85,B 0,C 180,E1 -5103.849,E2 -5103.849} C_VEL
LIN {X 0,Y 518.115,Z 300.628,A -85,B 0,C 180,E1 -5105.344,E2 -5105.344} C_VEL
LIN {X 0,Y 517.889,Z 312.026,A -85,B 0,C 180,E1 -5107.669,E2 -5107.669} C_VEL
LIN {X 0,Y 517.538,Z 325.606,A -85,B 0,C 180,E1 -5110.361,E2 -5110.361} C_VEL
LIN {X 0,Y 517.211,Z 340.146,A -85,B 0,C 180,E1 -5113.217,E2 -5113.217} C_VEL
LIN {X 0,Y 517.049,Z 347.306,A -85,B 0,C 180,E1 -5114.609,E2 -5114.609} C_VEL
LIN {X 0,Y 517.81,Z 352.282,A -85,B 0,C 180,E1 -5114.739,E2 -5114.739} C_VEL
LIN {X 0,Y 519.092,Z 360.444,A -85,B 0,C 180,E1 -5114.892,E2 -5114.892} C_VEL
LIN {X 0,Y 518.669,Z 452.294,A -85,B 0,C 180,E1 -5116.183,E2 -5116.183} C_VEL
LIN {X 0,Y 518.478,Z 462.186,A -85,B 0,C 180,E1 -5116.403,E2 -5116.403} C_VEL
LIN {X 0,Y 518.289,Z 472.162,A -85,B 0,C 180,E1 -5116.723,E2 -5116.723} C_VEL
LIN {X 0,Y 518.067,Z 481.519,A -85,B 0,C 180,E1 -5117.116,E2 -5117.116} C_VEL
LIN {X 0,Y 517.797,Z 492.156,A -85,B 0,C 180,E1 -5117.687,E2 -5117.687} C_VEL
LIN {X 0,Y 517.617,Z 500.663,A -85,B 0,C 180,E1 -5118.249,E2 -5118.249} C_VEL
LIN {X 0,Y 517.35,Z 509.394,A -85,B 0,C 180,E1 -5118.938,E2 -5118.938} C_VEL
LIN {X 0,Y 517.109,Z 516.79,A -85,B 0,C 180,E1 -5119.626,E2 -5119.626} C_VEL
LIN {X 0,Y 516.934,Z 524.012,A -85,B 0,C 180,E1 -5120.413,E2 -5120.413} C_VEL
LIN {X 0,Y 516.728,Z 530.214,A -85,B 0,C 180,E1 -5121.199,E2 -5121.199} C_VEL
LIN {X 0,Y 516.586,Z 536.751,A -85,B 0,C 180,E1 -5122.181,E2 -5122.181} C_VEL
LIN {X 0,Y 516.5,Z 541.252,A -85,B 0,C 180,E1 -5122.966,E2 -5122.966} C_VEL
LIN {X 0,Y 516.412,Z 546.741,A -85,B 0,C 180,E1 -5124.142,E2 -5124.142} C_VEL
LIN {X 0,Y 516.275,Z 551.059,A -85,B 0,C 180,E1 -5125.315,E2 -5125.315} C_VEL
LIN {X 0,Y 516.353,Z 553.425,A -85,B 0,C 180,E1 -5126.098,E2 -5126.098} C_VEL
LIN {X 0,Y 516.282,Z 555.219,A -85,B 0,C 180,E1 -5126.879,E2 -5126.879} C_VEL
LIN {X 0,Y 516.192,Z 557.656,A -85,B 0,C 180,E1 -5128.44,E2 -5128.44} C_VEL
LIN {X 0,Y 516.16,Z 558.242,A -85,B 0,C 180,E1 -5129.22,E2 -5129.22} C_VEL
LIN {X 0,Y 516.16,Z 558.242,A -85,B 0,C 180,E1 -5130.78,E2 -5130.78} C_VEL
LIN {X 0,Y 516.192,Z 557.656,A -85,B 0,C 180,E1 -5131.56,E2 -5131.56} C_VEL
LIN {X 0,Y 516.282,Z 555.219,A -85,B 0,C 180,E1 -5133.121,E2 -5133.121} C_VEL
LIN {X 0,Y 516.315,Z 552.275,A -85,B 0,C 180,E1 -5134.293,E2 -5134.293} C_VEL
LIN {X 0,Y 516.373,Z 548.293,A -85,B 0,C 180,E1 -5135.467,E2 -5135.467} C_VEL
LIN {X 0,Y 516.427,Z 543.572,A -85,B 0,C 180,E1 -5136.559,E2 -5136.559} C_VEL
LIN {X 0,Y 516.545,Z 537.906,A -85,B 0,C 180,E1 -5137.623,E2 -5137.623} C_VEL
LIN {X 0,Y 516.721,Z 531.591,A -85,B 0,C 180,E1 -5138.604,E2 -5138.604} C_VEL
LIN {X 0,Y 516.893,Z 525.639,A -85,B 0,C 180,E1 -5139.39,E2 -5139.39} C_VEL
LIN {X 0,Y 517.039,Z 518.71,A -85,B 0,C 180,E1 -5140.178,E2 -5140.178} C_VEL
LIN {X 0,Y 517.338,Z 510.53,A -85,B 0,C 180,E1 -5140.964,E2 -5140.964} C_VEL
LIN {X 0,Y 517.569,Z 502.015,A -85,B 0,C 180,E1 -5141.653,E2 -5141.653} C_VEL
LIN {X 0,Y 517.772,Z 493.506,A -85,B 0,C 180,E1 -5142.232,E2 -5142.232} C_VEL
LIN {X 0,Y 518.02,Z 483.534,A -85,B 0,C 180,E1 -5142.786,E2 -5142.786} C_VEL
LIN {X 0,Y 518.252,Z 474.738,A -85,B 0,C 180,E1 -5143.179,E2 -5143.179} C_VEL
LIN {X 0,Y 518.431,Z 464.809,A -85,B 0,C 180,E1 -5143.523,E2 -5143.523} C_VEL
LIN {X 0,Y 518.603,Z 454.957,A -85,B 0,C 180,E1 -5143.768,E2 -5143.768} C_VEL
LIN {X 0,Y 518.79,Z 430.352,A -85,B 0,C 180,E1 -5144.138,E2 -5144.138} C_VEL
LIN {X 0,Y 518.963,Z 358.901,A -85,B 0,C 180,E1 -5145.134,E2 -5145.134} C_VEL
LIN {X 0,Y 517.077,Z 347.514,A -85,B 0,C 180,E1 -5145.374,E2 -5145.374} C_VEL
LIN {X 0,Y 517.307,Z 335.488,A -85,B 0,C 180,E1 -5147.705,E2 -5147.705} C_VEL
LIN {X 0,Y 517.779,Z 318.285,A -85,B 0,C 180,E1 -5151.081,E2 -5151.081} C_VEL
LIN {X 0,Y 518.187,Z 302.2,A -85,B 0,C 180,E1 -5154.331,E2 -5154.331} C_VEL
LIN {X 0,Y 517.283,Z 295.507,A -85,B 0,C 180,E1 -5155.77,E2 -5155.77} C_VEL
LIN {X 0,Y 516.955,Z 293.609,A -85,B 0,C 180,E1 -5156.249,E2 -5156.249} C_VEL
LIN {X 0,Y 516.91,Z 293.597,A -85,B 0,C 180,E1 -5159.523,E2 -5159.523} C_VEL
LIN {X 0,Y 516.895,Z 293.595,A -85,B 0,C 180,E1 -5162.542,E2 -5162.542} C_VEL
LIN {X 0,Y 516.862,Z 293.599,A -85,B 0,C 180,E1 -5165.328,E2 -5165.328} C_VEL
LIN {X 0,Y 516.876,Z 293.605,A -85,B 0,C 180,E1 -5167.942,E2 -5167.942} C_VEL
LIN {X 0,Y 516.88,Z 293.589,A -85,B 0,C 180,E1 -5170.741,E2 -5170.741} C_VEL
LIN {X 0,Y 516.879,Z 293.596,A -85,B 0,C 180,E1 -5172.831,E2 -5172.831} C_VEL
LIN {X 0,Y 516.891,Z 293.594,A -85,B 0,C 180,E1 -5175.006,E2 -5175.006} C_VEL
LIN {X 0,Y 516.912,Z 293.592,A -85,B 0,C 180,E1 -5178.397,E2 -5178.397} C_VEL
LIN {X 0,Y 516.875,Z 293.596,A -85,B 0,C 180,E1 -5181.283,E2 -5181.283} C_VEL
LIN {X 0,Y 516.865,Z 293.597,A -85,B 0,C 180,E1 -5184.219,E2 -5184.219} C_VEL
LIN {X 0,Y 516.874,Z 293.593,A -85,B 0,C 180,E1 -5187.051,E2 -5187.051} C_VEL
LIN {X 0,Y 516.885,Z 293.601,A -85,B 0,C 180,E1 -5189.795,E2 -5189.795} C_VEL
LIN {X 0,Y 516.921,Z 293.584,A -85,B 0,C 180,E1 -5192.467,E2 -5192.467} C_VEL
LIN {X 0,Y 516.867,Z 293.595,A -85,B 0,C 180,E1 -5195.069,E2 -5195.069} C_VEL
LIN {X 0,Y 516.86,Z 293.604,A -85,B 0,C 180,E1 -5197.621,E2 -5197.621} C_VEL
LIN {X 0,Y 516.924,Z 293.584,A -85,B 0,C 180,E1 -5200.129,E2 -5200.129} C_VEL
LIN {X 0,Y 516.92,Z 293.583,A -85,B 0,C 180,E1 -5202.595,E2 -5202.595} C_VEL
LIN {X 0,Y 516.942,Z 293.589,A -85,B 0,C 180,E1 -5205.03,E2 -5205.03} C_VEL
LIN {X 0,Y 516.956,Z 293.582,A -85,B 0,C 180,E1 -5208.233,E2 -5208.233} C_VEL
LIN {X 0,Y 516.963,Z 293.583,A -85,B 0,C 180,E1 -5211.399,E2 -5211.399} C_VEL
LIN {X 0,Y 517,Z 293.583,A -85,B 0,C 180,E1 -5213.756,E2 -5213.756} C_VEL
LIN {X 0,Y 517.072,Z 293.571,A -85,B 0,C 180,E1 -5217.663,E2 -5217.663} C_VEL
LIN {X 0,Y 517.086,Z 293.561,A -85,B 0,C 180,E1 -5220.778,E2 -5220.778} C_VEL
LIN {X 0,Y 517.007,Z 293.583,A -85,B 0,C 180,E1 -5223.117,E2 -5223.117} C_VEL
LIN {X 0,Y 516.999,Z 293.58,A -85,B 0,C 180,E1 -5226.243,E2 -5226.243} C_VEL
LIN {X 0,Y 516.945,Z 293.581,A -85,B 0,C 180,E1 -5229.389,E2 -5229.389} C_VEL
LIN {X 0,Y 516.947,Z 293.584,A -85,B 0,C 180,E1 -5231.81,E2 -5231.81} C_VEL
LIN {X 0,Y 516.933,Z 293.595,A -85,B 0,C 180,E1 -5235.146,E2 -5235.146} C_VEL
LIN {X 0,Y 516.914,Z 293.586,A -85,B 0,C 180,E1 -5238.222,E2 -5238.222} C_VEL
LIN {X 0,Y 516.902,Z 293.591,A -85,B 0,C 180,E1 -5240.701,E2 -5240.701} C_VEL
LIN {X 0,Y 516.901,Z 293.593,A -85,B 0,C 180,E1 -5244.072,E2 -5244.072} C_VEL
LIN {X 0,Y 516.916,Z 293.594,A -85,B 0,C 180,E1 -5246.658,E2 -5246.658} C_VEL
LIN {X 0,Y 516.915,Z 293.591,A -85,B 0,C 180,E1 -5249.527,E2 -5249.527} C_VEL
LIN {X 0,Y 516.891,Z 293.6,A -85,B 0,C 180,E1 -5252.545,E2 -5252.545} C_VEL
LIN {X 0,Y 516.874,Z 293.595,A -85,B 0,C 180,E1 -5255.333,E2 -5255.333} C_VEL
LIN {X 0,Y 516.872,Z 293.597,A -85,B 0,C 180,E1 -5257.944,E2 -5257.944} C_VEL
LIN {X 0,Y 516.895,Z 293.597,A -85,B 0,C 180,E1 -5260.74,E2 -5260.74} C_VEL
LIN {X 0,Y 516.874,Z 293.597,A -85,B 0,C 180,E1 -5263.903,E2 -5263.903} C_VEL
LIN {X 0,Y 516.874,Z 293.595,A -85,B 0,C 180,E1 -5266.107,E2 -5266.107} C_VEL
LIN {X 0,Y 516.909,Z 293.582,A -85,B 0,C 180,E1 -5268.399,E2 -5268.399} C_VEL
LIN {X 0,Y 516.874,Z 293.596,A -85,B 0,C 180,E1 -5270.314,E2 -5270.314} C_VEL
LIN {X 0,Y 516.205,Z 293.685,A -85,B 0,C 180,E1 -5270.964,E2 -5270.964} C_VEL
LIN {X 0,Y 513.359,Z 294.039,A -85,B 0,C 180,E1 -5272.02,E2 -5272.02} C_VEL
LIN {X 0,Y 510.951,Z 294.337,A -85,B 0,C 180,E1 -5272.87,E2 -5272.87} C_VEL
LIN {X 0,Y 509.912,Z 294.463,A -85,B 0,C 180,E1 -5273.527,E2 -5273.527} C_VEL
LIN {X 0,Y 509.824,Z 294.473,A -85,B 0,C 180,E1 -5273.749,E2 -5273.749} C_VEL
LIN {X 0,Y 509.857,Z 294.471,A -85,B 0,C 180,E1 -5276.54,E2 -5276.54} C_VEL
LIN {X 0,Y 509.84,Z 294.472,A -85,B 0,C 180,E1 -5279.335,E2 -5279.335} C_VEL
LIN {X 0,Y 509.889,Z 294.468,A -85,B 0,C 180,E1 -5282.055,E2 -5282.055} C_VEL
LIN {X 0,Y 509.873,Z 294.474,A -85,B 0,C 180,E1 -5284.704,E2 -5284.704} C_VEL
LIN {X 0,Y 509.832,Z 294.475,A -85,B 0,C 180,E1 -5287.455,E2 -5287.455} C_VEL
LIN {X 0,Y 509.912,Z 294.468,A -85,B 0,C 180,E1 -5289.845,E2 -5289.845} C_VEL
LIN {X 0,Y 509.882,Z 294.469,A -85,B 0,C 180,E1 -5293.175,E2 -5293.175} C_VEL
LIN {X 0,Y 509.86,Z 294.474,A -85,B 0,C 180,E1 -5295.634,E2 -5295.634} C_VEL
LIN {X 0,Y 509.91,Z 294.467,A -85,B 0,C 180,E1 -5298.875,E2 -5298.875} C_VEL
LIN {X 0,Y 509.948,Z 294.468,A -85,B 0,C 180,E1 -5302.079,E2 -5302.079} C_VEL
LIN {X 0,Y 509.98,Z 294.461,A -85,B 0,C 180,E1 -5304.464,E2 -5304.464} C_VEL
LIN {X 0,Y 510.053,Z 294.452,A -85,B 0,C 180,E1 -5307.631,E2 -5307.631} C_VEL
LIN {X 0,Y 510.061,Z 294.448,A -85,B 0,C 180,E1 -5310.789,E2 -5310.789} C_VEL
LIN {X 0,Y 509.952,Z 294.461,A -85,B 0,C 180,E1 -5313.16,E2 -5313.16} C_VEL
LIN {X 0,Y 509.977,Z 294.461,A -85,B 0,C 180,E1 -5316.329,E2 -5316.329} C_VEL
LIN {X 0,Y 509.912,Z 294.466,A -85,B 0,C 180,E1 -5318.72,E2 -5318.72} C_VEL
LIN {X 0,Y 509.9,Z 294.473,A -85,B 0,C 180,E1 -5321.931,E2 -5321.931} C_VEL
LIN {X 0,Y 509.889,Z 294.471,A -85,B 0,C 180,E1 -5325.242,E2 -5325.242} C_VEL
LIN {X 0,Y 509.884,Z 294.474,A -85,B 0,C 180,E1 -5328.001,E2 -5328.001} C_VEL
LIN {X 0,Y 509.846,Z 294.474,A -85,B 0,C 180,E1 -5331.001,E2 -5331.001} C_VEL
LIN {X 0,Y 509.832,Z 294.482,A -85,B 0,C 180,E1 -5333.563,E2 -5333.563} C_VEL
LIN {X 0,Y 509.908,Z 294.466,A -85,B 0,C 180,E1 -5336.379,E2 -5336.379} C_VEL
LIN {X 0,Y 509.872,Z 294.466,A -85,B 0,C 180,E1 -5338.844,E2 -5338.844} C_VEL
LIN {X 0,Y 509.82,Z 294.484,A -85,B 0,C 180,E1 -5341.589,E2 -5341.589} C_VEL
LIN {X 0,Y 509.848,Z 294.461,A -85,B 0,C 180,E1 -5344.413,E2 -5344.413} C_VEL
LIN {X 0,Y 509.812,Z 294.481,A -85,B 0,C 180,E1 -5347.34,E2 -5347.34} C_VEL
LIN {X 0,Y 509.831,Z 294.468,A -85,B 0,C 180,E1 -5350.382,E2 -5350.382} C_VEL
LIN {X 0,Y 509.831,Z 294.463,A -85,B 0,C 180,E1 -5353.064,E2 -5353.064} C_VEL
LIN {X 0,Y 509.822,Z 294.478,A -85,B 0,C 180,E1 -5355.792,E2 -5355.792} C_VEL
LIN {X 0,Y 509.856,Z 294.469,A -85,B 0,C 180,E1 -5358.575,E2 -5358.575} C_VEL
LIN {X 0,Y 509.843,Z 294.475,A -85,B 0,C 180,E1 -5361.786,E2 -5361.786} C_VEL
LIN {X 0,Y 509.837,Z 294.472,A -85,B 0,C 180,E1 -5364.623,E2 -5364.623} C_VEL
LIN {X 0,Y 509.856,Z 294.476,A -85,B 0,C 180,E1 -5367.481,E2 -5367.481} C_VEL
LIN {X 0,Y 509.872,Z 294.468,A -85,B 0,C 180,E1 -5370.269,E2 -5370.269} C_VEL
LIN {X 0,Y 509.875,Z 294.466,A -85,B 0,C 180,E1 -5372.944,E2 -5372.944} C_VEL
LIN {X 0,Y 509.859,Z 294.473,A -85,B 0,C 180,E1 -5375.574,E2 -5375.574} C_VEL
LIN {X 0,Y 509.812,Z 294.475,A -85,B 0,C 180,E1 -5378.149,E2 -5378.149} C_VEL
LIN {X 0,Y 509.855,Z 294.467,A -85,B 0,C 180,E1 -5380.682,E2 -5380.682} C_VEL
LIN {X 0,Y 509.877,Z 294.473,A -85,B 0,C 180,E1 -5383.175,E2 -5383.175} C_VEL
LIN {X 0,Y 509.853,Z 294.472,A -85,B 0,C 180,E1 -5385.634,E2 -5385.634} C_VEL
LIN {X 0,Y 509.907,Z 294.462,A -85,B 0,C 180,E1 -5388.875,E2 -5388.875} C_VEL
LIN {X 0,Y 509.941,Z 294.455,A -85,B 0,C 180,E1 -5392.079,E2 -5392.079} C_VEL
LIN {X 0,Y 509.973,Z 294.459,A -85,B 0,C 180,E1 -5394.465,E2 -5394.465} C_VEL
LIN {X 0,Y 510.044,Z 294.442,A -85,B 0,C 180,E1 -5397.631,E2 -5397.631} C_VEL
LIN {X 0,Y 510.057,Z 294.442,A -85,B 0,C 180,E1 -5400.79,E2 -5400.79} C_VEL
LIN {X 0,Y 509.948,Z 294.462,A -85,B 0,C 180,E1 -5403.161,E2 -5403.161} C_VEL
LIN {X 0,Y 509.968,Z 294.46,A -85,B 0,C 180,E1 -5406.33,E2 -5406.33} C_VEL
LIN {X 0,Y 509.909,Z 294.459,A -85,B 0,C 180,E1 -5408.721,E2 -5408.721} C_VEL
LIN {X 0,Y 509.896,Z 294.462,A -85,B 0,C 180,E1 -5411.932,E2 -5411.932} C_VEL
LIN {X 0,Y 509.885,Z 294.466,A -85,B 0,C 180,E1 -5415.242,E2 -5415.242} C_VEL
LIN {X 0,Y 509.88,Z 294.462,A -85,B 0,C 180,E1 -5418.002,E2 -5418.002} C_VEL
LIN {X 0,Y 509.843,Z 294.473,A -85,B 0,C 180,E1 -5421.002,E2 -5421.002} C_VEL
LIN {X 0,Y 509.815,Z 294.475,A -85,B 0,C 180,E1 -5423.565,E2 -5423.565} C_VEL
LIN {X 0,Y 509.904,Z 294.464,A -85,B 0,C 180,E1 -5426.379,E2 -5426.379} C_VEL
LIN {X 0,Y 509.87,Z 294.471,A -85,B 0,C 180,E1 -5428.845,E2 -5428.845} C_VEL
LIN {X 0,Y 509.813,Z 294.476,A -85,B 0,C 180,E1 -5431.591,E2 -5431.591} C_VEL
LIN {X 0,Y 509.832,Z 294.475,A -85,B 0,C 180,E1 -5434.415,E2 -5434.415} C_VEL
LIN {X 0,Y 509.811,Z 294.476,A -85,B 0,C 180,E1 -5437.342,E2 -5437.342} C_VEL
LIN {X 0,Y 509.833,Z 294.478,A -85,B 0,C 180,E1 -5440.383,E2 -5440.383} C_VEL
LIN {X 0,Y 509.818,Z 294.475,A -85,B 0,C 180,E1 -5443.063,E2 -5443.063} C_VEL
LIN {X 0,Y 509.818,Z 294.478,A -85,B 0,C 180,E1 -5445.794,E2 -5445.794} C_VEL
LIN {X 0,Y 509.852,Z 294.466,A -85,B 0,C 180,E1 -5448.575,E2 -5448.575} C_VEL
LIN {X 0,Y 509.847,Z 294.476,A -85,B 0,C 180,E1 -5451.788,E2 -5451.788} C_VEL
LIN {X 0,Y 509.826,Z 294.475,A -85,B 0,C 180,E1 -5454.623,E2 -5454.623} C_VEL
LIN {X 0,Y 509.86,Z 294.472,A -85,B 0,C 180,E1 -5457.482,E2 -5457.482} C_VEL
LIN {X 0,Y 509.858,Z 294.475,A -85,B 0,C 180,E1 -5460.275,E2 -5460.275} C_VEL
LIN {X 0,Y 509.89,Z 294.471,A -85,B 0,C 180,E1 -5463.325,E2 -5463.325} C_VEL
LIN {X 0,Y 509.951,Z 294.673,A -85,B 0,C 180,E1 -5463.663,E2 -5463.663} C_VEL
LIN {X 0,Y 511.202,Z 302.504,A -85,B 0,C 180,E1 -5465.408,E2 -5465.408} C_VEL
LIN {X 0,Y 510.843,Z 316.055,A -85,B 0,C 180,E1 -5468.195,E2 -5468.195} C_VEL
LIN {X 0,Y 510.415,Z 332.754,A -85,B 0,C 180,E1 -5471.538,E2 -5471.538} C_VEL
LIN {X 0,Y 510.024,Z 347.103,A -85,B 0,C 180,E1 -5474.39,E2 -5474.39} C_VEL
LIN {X 0,Y 510.763,Z 351.826,A -85,B 0,C 180,E1 -5474.52,E2 -5474.52} C_VEL
LIN {X 0,Y 512.238,Z 361.397,A -85,B 0,C 180,E1 -5474.701,E2 -5474.701} C_VEL
LIN {X 0,Y 511.79,Z 452.101,A -85,B 0,C 180,E1 -5475.994,E2 -5475.994} C_VEL
LIN {X 0,Y 511.575,Z 461.992,A -85,B 0,C 180,E1 -5476.216,E2 -5476.216} C_VEL
LIN {X 0,Y 511.387,Z 471.968,A -85,B 0,C 180,E1 -5476.54,E2 -5476.54} C_VEL
LIN {X 0,Y 511.113,Z 481.324,A -85,B 0,C 180,E1 -5476.937,E2 -5476.937} C_VEL
LIN {X 0,Y 510.862,Z 491.808,A -85,B 0,C 180,E1 -5477.507,E2 -5477.507} C_VEL
LIN {X 0,Y 510.64,Z 500.469,A -85,B 0,C 180,E1 -5478.086,E2 -5478.086} C_VEL
LIN {X 0,Y 510.349,Z 509.199,A -85,B 0,C 180,E1 -5478.784,E2 -5478.784} C_VEL
LIN {X 0,Y 510.081,Z 516.595,A -85,B 0,C 180,E1 -5479.481,E2 -5479.481} C_VEL
LIN {X 0,Y 509.879,Z 523.817,A -85,B 0,C 180,E1 -5480.279,E2 -5480.279} C_VEL
LIN {X 0,Y 509.682,Z 530.019,A -85,B 0,C 180,E1 -5481.076,E2 -5481.076} C_VEL
LIN {X 0,Y 509.527,Z 536.557,A -85,B 0,C 180,E1 -5482.072,E2 -5482.072} C_VEL
LIN {X 0,Y 509.397,Z 542.111,A -85,B 0,C 180,E1 -5483.086,E2 -5483.086} C_VEL
LIN {X 0,Y 509.307,Z 546.546,A -85,B 0,C 180,E1 -5484.06,E2 -5484.06} C_VEL
LIN {X 0,Y 509.192,Z 550.865,A -85,B 0,C 180,E1 -5485.25,E2 -5485.25} C_VEL
LIN {X 0,Y 509.246,Z 553.23,A -85,B 0,C 180,E1 -5486.043,E2 -5486.043} C_VEL
LIN {X 0,Y 509.201,Z 555.025,A -85,B 0,C 180,E1 -5486.835,E2 -5486.835} C_VEL
LIN {X 0,Y 509.113,Z 557.462,A -85,B 0,C 180,E1 -5488.418,E2 -5488.418} C_VEL
LIN {X 0,Y 509.074,Z 558.048,A -85,B 0,C 180,E1 -5489.209,E2 -5489.209} C_VEL
LIN {X 0,Y 509.074,Z 558.048,A -85,B 0,C 180,E1 -5490.791,E2 -5490.791} C_VEL
LIN {X 0,Y 509.113,Z 557.462,A -85,B 0,C 180,E1 -5491.582,E2 -5491.582} C_VEL
LIN {X 0,Y 509.201,Z 555.025,A -85,B 0,C 180,E1 -5493.165,E2 -5493.165} C_VEL
LIN {X 0,Y 509.207,Z 552.081,A -85,B 0,C 180,E1 -5494.353,E2 -5494.353} C_VEL
LIN {X 0,Y 509.29,Z 548.099,A -85,B 0,C 180,E1 -5495.543,E2 -5495.543} C_VEL
LIN {X 0,Y 509.35,Z 543.831,A -85,B 0,C 180,E1 -5496.557,E2 -5496.557} C_VEL
